//     Term 19 (AT2200-0500)/CC Outputs/Current setpoint value Ch.8 <-> Data Pointer/CurrentSetpointValues[7]
//     Term 19 (AT2200-0500)/CC Outputs/Current setpoint value Ch.9 <-> Data Pointer/CurrentSetpointValues[8]
//     Term 19 (AT2200-0500)/LFB Inputs/BinaryData <-> Data Pointer/HallSensorValues
//   Device 20 <-> TcCOM Objects/XTS ProcessingUnit 1/Part 1/Module 16
//     Term 20 (AT2200-0500)/CC Inputs/Current actual value Ch.1 <-> Data Pointer/CurrentActualValues[0]
//     Term 20 (AT2200-0500)/CC Inputs/Current actual value Ch.10 <-> Data Pointer/CurrentActualValues[9]
//     Term 20 (AT2200-0500)/CC Inputs/Current actual value Ch.11 <-> Data Pointer/CurrentActualValues[10]
//     Term 20 (AT2200-0500)/CC Inputs/Current actual value Ch.12 <-> Data Pointer/CurrentActualValues[11]
//     Term 20 (AT2200-0500)/CC Inputs/Current actual value Ch.13 <-> Data Pointer/CurrentActualValues[12]
//     Term 20 (AT2200-0500)/CC Inputs/Current actual value Ch.14 <-> Data Pointer/CurrentActualValues[13]
//     Term 20 (AT2200-0500)/CC Inputs/Current actual value Ch.15 <-> Data Pointer/CurrentActualValues[14]
//     Term 20 (AT2200-0500)/CC Inputs/Current actual value Ch.16 <-> Data Pointer/CurrentActualValues[15]
//     Term 20 (AT2200-0500)/CC Inputs/Current actual value Ch.17 <-> Data Pointer/CurrentActualValues[16]
//     Term 20 (AT2200-0500)/CC Inputs/Current actual value Ch.18 <-> Data Pointer/CurrentActualValues[17]
//     Term 20 (AT2200-0500)/CC Inputs/Current actual value Ch.19 <-> Data Pointer/CurrentActualValues[18]
//     Term 20 (AT2200-0500)/CC Inputs/Current actual value Ch.2 <-> Data Pointer/CurrentActualValues[1]
//     Term 20 (AT2200-0500)/CC Inputs/Current actual value Ch.20 <-> Data Pointer/CurrentActualValues[19]
//     Term 20 (AT2200-0500)/CC Inputs/Current actual value Ch.21 <-> Data Pointer/CurrentActualValues[20]
//     Term 20 (AT2200-0500)/CC Inputs/Current actual value Ch.22 <-> Data Pointer/CurrentActualValues[21]
//     Term 20 (AT2200-0500)/CC Inputs/Current actual value Ch.23 <-> Data Pointer/CurrentActualValues[22]
//     Term 20 (AT2200-0500)/CC Inputs/Current actual value Ch.24 <-> Data Pointer/CurrentActualValues[23]
//     Term 20 (AT2200-0500)/CC Inputs/Current actual value Ch.25 <-> Data Pointer/CurrentActualValues[24]
//     Term 20 (AT2200-0500)/CC Inputs/Current actual value Ch.26 <-> Data Pointer/CurrentActualValues[25]
//     Term 20 (AT2200-0500)/CC Inputs/Current actual value Ch.27 <-> Data Pointer/CurrentActualValues[26]
//     Term 20 (AT2200-0500)/CC Inputs/Current actual value Ch.28 <-> Data Pointer/CurrentActualValues[27]
//     Term 20 (AT2200-0500)/CC Inputs/Current actual value Ch.29 <-> Data Pointer/CurrentActualValues[28]
//     Term 20 (AT2200-0500)/CC Inputs/Current actual value Ch.3 <-> Data Pointer/CurrentActualValues[2]
//     Term 20 (AT2200-0500)/CC Inputs/Current actual value Ch.30 <-> Data Pointer/CurrentActualValues[29]
//     Term 20 (AT2200-0500)/CC Inputs/Current actual value Ch.4 <-> Data Pointer/CurrentActualValues[3]
//     Term 20 (AT2200-0500)/CC Inputs/Current actual value Ch.5 <-> Data Pointer/CurrentActualValues[4]
//     Term 20 (AT2200-0500)/CC Inputs/Current actual value Ch.6 <-> Data Pointer/CurrentActualValues[5]
//     Term 20 (AT2200-0500)/CC Inputs/Current actual value Ch.7 <-> Data Pointer/CurrentActualValues[6]
//     Term 20 (AT2200-0500)/CC Inputs/Current actual value Ch.8 <-> Data Pointer/CurrentActualValues[7]
//     Term 20 (AT2200-0500)/CC Inputs/Current actual value Ch.9 <-> Data Pointer/CurrentActualValues[8]
//     Term 20 (AT2200-0500)/CC Inputs/Status <-> Data Pointer/Status
//     Term 20 (AT2200-0500)/CC Outputs/Control <-> Data Pointer/Control
//     Term 20 (AT2200-0500)/CC Outputs/Current setpoint value Ch.1 <-> Data Pointer/CurrentSetpointValues[0]
//     Term 20 (AT2200-0500)/CC Outputs/Current setpoint value Ch.10 <-> Data Pointer/CurrentSetpointValues[9]
//     Term 20 (AT2200-0500)/CC Outputs/Current setpoint value Ch.11 <-> Data Pointer/CurrentSetpointValues[10]
//     Term 20 (AT2200-0500)/CC Outputs/Current setpoint value Ch.12 <-> Data Pointer/CurrentSetpointValues[11]
//     Term 20 (AT2200-0500)/CC Outputs/Current setpoint value Ch.13 <-> Data Pointer/CurrentSetpointValues[12]
//     Term 20 (AT2200-0500)/CC Outputs/Current setpoint value Ch.14 <-> Data Pointer/CurrentSetpointValues[13]
//     Term 20 (AT2200-0500)/CC Outputs/Current setpoint value Ch.15 <-> Data Pointer/CurrentSetpointValues[14]
//     Term 20 (AT2200-0500)/CC Outputs/Current setpoint value Ch.16 <-> Data Pointer/CurrentSetpointValues[15]
//     Term 20 (AT2200-0500)/CC Outputs/Current setpoint value Ch.17 <-> Data Pointer/CurrentSetpointValues[16]
//     Term 20 (AT2200-0500)/CC Outputs/Current setpoint value Ch.18 <-> Data Pointer/CurrentSetpointValues[17]
//     Term 20 (AT2200-0500)/CC Outputs/Current setpoint value Ch.19 <-> Data Pointer/CurrentSetpointValues[18]
//     Term 20 (AT2200-0500)/CC Outputs/Current setpoint value Ch.2 <-> Data Pointer/CurrentSetpointValues[1]
//     Term 20 (AT2200-0500)/CC Outputs/Current setpoint value Ch.20 <-> Data Pointer/CurrentSetpointValues[19]
//     Term 20 (AT2200-0500)/CC Outputs/Current setpoint value Ch.21 <-> Data Pointer/CurrentSetpointValues[20]
//     Term 20 (AT2200-0500)/CC Outputs/Current setpoint value Ch.22 <-> Data Pointer/CurrentSetpointValues[21]
//     Term 20 (AT2200-0500)/CC Outputs/Current setpoint value Ch.23 <-> Data Pointer/CurrentSetpointValues[22]
//     Term 20 (AT2200-0500)/CC Outputs/Current setpoint value Ch.24 <-> Data Pointer/CurrentSetpointValues[23]
//     Term 20 (AT2200-0500)/CC Outputs/Current setpoint value Ch.25 <-> Data Pointer/CurrentSetpointValues[24]
//     Term 20 (AT2200-0500)/CC Outputs/Current setpoint value Ch.26 <-> Data Pointer/CurrentSetpointValues[25]
//     Term 20 (AT2200-0500)/CC Outputs/Current setpoint value Ch.27 <-> Data Pointer/CurrentSetpointValues[26]
//     Term 20 (AT2200-0500)/CC Outputs/Current setpoint value Ch.28 <-> Data Pointer/CurrentSetpointValues[27]
//     Term 20 (AT2200-0500)/CC Outputs/Current setpoint value Ch.29 <-> Data Pointer/CurrentSetpointValues[28]
//     Term 20 (AT2200-0500)/CC Outputs/Current setpoint value Ch.3 <-> Data Pointer/CurrentSetpointValues[2]
//     Term 20 (AT2200-0500)/CC Outputs/Current setpoint value Ch.30 <-> Data Pointer/CurrentSetpointValues[29]
//     Term 20 (AT2200-0500)/CC Outputs/Current setpoint value Ch.4 <-> Data Pointer/CurrentSetpointValues[3]
//     Term 20 (AT2200-0500)/CC Outputs/Current setpoint value Ch.5 <-> Data Pointer/CurrentSetpointValues[4]
//     Term 20 (AT2200-0500)/CC Outputs/Current setpoint value Ch.6 <-> Data Pointer/CurrentSetpointValues[5]
//     Term 20 (AT2200-0500)/CC Outputs/Current setpoint value Ch.7 <-> Data Pointer/CurrentSetpointValues[6]
//     Term 20 (AT2200-0500)/CC Outputs/Current setpoint value Ch.8 <-> Data Pointer/CurrentSetpointValues[7]
//     Term 20 (AT2200-0500)/CC Outputs/Current setpoint value Ch.9 <-> Data Pointer/CurrentSetpointValues[8]
//     Term 20 (AT2200-0500)/LFB Inputs/BinaryData <-> Data Pointer/HallSensorValues
//   Device 21 <-> TcCOM Objects/XTS ProcessingUnit 1/Part 1/Module 17
//     Term 21 (AT2202-0500)/CC Inputs/Current actual value Ch.1 <-> Data Pointer/CurrentActualValues[0]
//     Term 21 (AT2202-0500)/CC Inputs/Current actual value Ch.10 <-> Data Pointer/CurrentActualValues[9]
//     Term 21 (AT2202-0500)/CC Inputs/Current actual value Ch.11 <-> Data Pointer/CurrentActualValues[10]
//     Term 21 (AT2202-0500)/CC Inputs/Current actual value Ch.12 <-> Data Pointer/CurrentActualValues[11]
//     Term 21 (AT2202-0500)/CC Inputs/Current actual value Ch.13 <-> Data Pointer/CurrentActualValues[12]
//     Term 21 (AT2202-0500)/CC Inputs/Current actual value Ch.14 <-> Data Pointer/CurrentActualValues[13]
//     Term 21 (AT2202-0500)/CC Inputs/Current actual value Ch.15 <-> Data Pointer/CurrentActualValues[14]
//     Term 21 (AT2202-0500)/CC Inputs/Current actual value Ch.16 <-> Data Pointer/CurrentActualValues[15]
//     Term 21 (AT2202-0500)/CC Inputs/Current actual value Ch.17 <-> Data Pointer/CurrentActualValues[16]
//     Term 21 (AT2202-0500)/CC Inputs/Current actual value Ch.18 <-> Data Pointer/CurrentActualValues[17]
//     Term 21 (AT2202-0500)/CC Inputs/Current actual value Ch.19 <-> Data Pointer/CurrentActualValues[18]
//     Term 21 (AT2202-0500)/CC Inputs/Current actual value Ch.2 <-> Data Pointer/CurrentActualValues[1]
//     Term 21 (AT2202-0500)/CC Inputs/Current actual value Ch.20 <-> Data Pointer/CurrentActualValues[19]
//     Term 21 (AT2202-0500)/CC Inputs/Current actual value Ch.21 <-> Data Pointer/CurrentActualValues[20]
//     Term 21 (AT2202-0500)/CC Inputs/Current actual value Ch.22 <-> Data Pointer/CurrentActualValues[21]
//     Term 21 (AT2202-0500)/CC Inputs/Current actual value Ch.23 <-> Data Pointer/CurrentActualValues[22]
//     Term 21 (AT2202-0500)/CC Inputs/Current actual value Ch.24 <-> Data Pointer/CurrentActualValues[23]
//     Term 21 (AT2202-0500)/CC Inputs/Current actual value Ch.25 <-> Data Pointer/CurrentActualValues[24]
//     Term 21 (AT2202-0500)/CC Inputs/Current actual value Ch.26 <-> Data Pointer/CurrentActualValues[25]
//     Term 21 (AT2202-0500)/CC Inputs/Current actual value Ch.27 <-> Data Pointer/CurrentActualValues[26]
//     Term 21 (AT2202-0500)/CC Inputs/Current actual value Ch.28 <-> Data Pointer/CurrentActualValues[27]
//     Term 21 (AT2202-0500)/CC Inputs/Current actual value Ch.29 <-> Data Pointer/CurrentActualValues[28]
//     Term 21 (AT2202-0500)/CC Inputs/Current actual value Ch.3 <-> Data Pointer/CurrentActualValues[2]
//     Term 21 (AT2202-0500)/CC Inputs/Current actual value Ch.30 <-> Data Pointer/CurrentActualValues[29]
//     Term 21 (AT2202-0500)/CC Inputs/Current actual value Ch.4 <-> Data Pointer/CurrentActualValues[3]
//     Term 21 (AT2202-0500)/CC Inputs/Current actual value Ch.5 <-> Data Pointer/CurrentActualValues[4]
//     Term 21 (AT2202-0500)/CC Inputs/Current actual value Ch.6 <-> Data Pointer/CurrentActualValues[5]
//     Term 21 (AT2202-0500)/CC Inputs/Current actual value Ch.7 <-> Data Pointer/CurrentActualValues[6]
//     Term 21 (AT2202-0500)/CC Inputs/Current actual value Ch.8 <-> Data Pointer/CurrentActualValues[7]
//     Term 21 (AT2202-0500)/CC Inputs/Current actual value Ch.9 <-> Data Pointer/CurrentActualValues[8]
//     Term 21 (AT2202-0500)/CC Inputs/Status <-> Data Pointer/Status
//     Term 21 (AT2202-0500)/CC Outputs/Control <-> Data Pointer/Control
//     Term 21 (AT2202-0500)/CC Outputs/Current setpoint value Ch.1 <-> Data Pointer/CurrentSetpointValues[0]
//     Term 21 (AT2202-0500)/CC Outputs/Current setpoint value Ch.10 <-> Data Pointer/CurrentSetpointValues[9]
//     Term 21 (AT2202-0500)/CC Outputs/Current setpoint value Ch.11 <-> Data Pointer/CurrentSetpointValues[10]
//     Term 21 (AT2202-0500)/CC Outputs/Current setpoint value Ch.12 <-> Data Pointer/CurrentSetpointValues[11]
//     Term 21 (AT2202-0500)/CC Outputs/Current setpoint value Ch.13 <-> Data Pointer/CurrentSetpointValues[12]
//     Term 21 (AT2202-0500)/CC Outputs/Current setpoint value Ch.14 <-> Data Pointer/CurrentSetpointValues[13]
//     Term 21 (AT2202-0500)/CC Outputs/Current setpoint value Ch.15 <-> Data Pointer/CurrentSetpointValues[14]
//     Term 21 (AT2202-0500)/CC Outputs/Current setpoint value Ch.16 <-> Data Pointer/CurrentSetpointValues[15]
//     Term 21 (AT2202-0500)/CC Outputs/Current setpoint value Ch.17 <-> Data Pointer/CurrentSetpointValues[16]
//     Term 21 (AT2202-0500)/CC Outputs/Current setpoint value Ch.18 <-> Data Pointer/CurrentSetpointValues[17]
//     Term 21 (AT2202-0500)/CC Outputs/Current setpoint value Ch.19 <-> Data Pointer/CurrentSetpointValues[18]
//     Term 21 (AT2202-0500)/CC Outputs/Current setpoint value Ch.2 <-> Data Pointer/CurrentSetpointValues[1]
//     Term 21 (AT2202-0500)/CC Outputs/Current setpoint value Ch.20 <-> Data Pointer/CurrentSetpointValues[19]
//     Term 21 (AT2202-0500)/CC Outputs/Current setpoint value Ch.21 <-> Data Pointer/CurrentSetpointValues[20]
//     Term 21 (AT2202-0500)/CC Outputs/Current setpoint value Ch.22 <-> Data Pointer/CurrentSetpointValues[21]
//     Term 21 (AT2202-0500)/CC Outputs/Current setpoint value Ch.23 <-> Data Pointer/CurrentSetpointValues[22]
//     Term 21 (AT2202-0500)/CC Outputs/Current setpoint value Ch.24 <-> Data Pointer/CurrentSetpointValues[23]
//     Term 21 (AT2202-0500)/CC Outputs/Current setpoint value Ch.25 <-> Data Pointer/CurrentSetpointValues[24]
//     Term 21 (AT2202-0500)/CC Outputs/Current setpoint value Ch.26 <-> Data Pointer/CurrentSetpointValues[25]
//     Term 21 (AT2202-0500)/CC Outputs/Current setpoint value Ch.27 <-> Data Pointer/CurrentSetpointValues[26]
//     Term 21 (AT2202-0500)/CC Outputs/Current setpoint value Ch.28 <-> Data Pointer/CurrentSetpointValues[27]
//     Term 21 (AT2202-0500)/CC Outputs/Current setpoint value Ch.29 <-> Data Pointer/CurrentSetpointValues[28]
//     Term 21 (AT2202-0500)/CC Outputs/Current setpoint value Ch.3 <-> Data Pointer/CurrentSetpointValues[2]
//     Term 21 (AT2202-0500)/CC Outputs/Current setpoint value Ch.30 <-> Data Pointer/CurrentSetpointValues[29]
//     Term 21 (AT2202-0500)/CC Outputs/Current setpoint value Ch.4 <-> Data Pointer/CurrentSetpointValues[3]
//     Term 21 (AT2202-0500)/CC Outputs/Current setpoint value Ch.5 <-> Data Pointer/CurrentSetpointValues[4]
//     Term 21 (AT2202-0500)/CC Outputs/Current setpoint value Ch.6 <-> Data Pointer/CurrentSetpointValues[5]
//     Term 21 (AT2202-0500)/CC Outputs/Current setpoint value Ch.7 <-> Data Pointer/CurrentSetpointValues[6]
//     Term 21 (AT2202-0500)/CC Outputs/Current setpoint value Ch.8 <-> Data Pointer/CurrentSetpointValues[7]
//     Term 21 (AT2202-0500)/CC Outputs/Current setpoint value Ch.9 <-> Data Pointer/CurrentSetpointValues[8]
//     Term 21 (AT2202-0500)/LFB Inputs/BinaryData <-> Data Pointer/HallSensorValues
//   Device 21 <-> TcCOM Objects/XTS ProcessingUnit 1/Part 1/Module 18
//     Term 22 (AT2200-0500)/CC Inputs/Current actual value Ch.1 <-> Data Pointer/CurrentActualValues[0]
//     Term 22 (AT2200-0500)/CC Inputs/Current actual value Ch.10 <-> Data Pointer/CurrentActualValues[9]
//     Term 22 (AT2200-0500)/CC Inputs/Current actual value Ch.11 <-> Data Pointer/CurrentActualValues[10]
//     Term 22 (AT2200-0500)/CC Inputs/Current actual value Ch.12 <-> Data Pointer/CurrentActualValues[11]
//     Term 22 (AT2200-0500)/CC Inputs/Current actual value Ch.13 <-> Data Pointer/CurrentActualValues[12]
//     Term 22 (AT2200-0500)/CC Inputs/Current actual value Ch.14 <-> Data Pointer/CurrentActualValues[13]
//     Term 22 (AT2200-0500)/CC Inputs/Current actual value Ch.15 <-> Data Pointer/CurrentActualValues[14]
//     Term 22 (AT2200-0500)/CC Inputs/Current actual value Ch.16 <-> Data Pointer/CurrentActualValues[15]
//     Term 22 (AT2200-0500)/CC Inputs/Current actual value Ch.17 <-> Data Pointer/CurrentActualValues[16]
//     Term 22 (AT2200-0500)/CC Inputs/Current actual value Ch.18 <-> Data Pointer/CurrentActualValues[17]
//     Term 22 (AT2200-0500)/CC Inputs/Current actual value Ch.19 <-> Data Pointer/CurrentActualValues[18]
//     Term 22 (AT2200-0500)/CC Inputs/Current actual value Ch.2 <-> Data Pointer/CurrentActualValues[1]
//     Term 22 (AT2200-0500)/CC Inputs/Current actual value Ch.20 <-> Data Pointer/CurrentActualValues[19]
//     Term 22 (AT2200-0500)/CC Inputs/Current actual value Ch.21 <-> Data Pointer/CurrentActualValues[20]
//     Term 22 (AT2200-0500)/CC Inputs/Current actual value Ch.22 <-> Data Pointer/CurrentActualValues[21]
//     Term 22 (AT2200-0500)/CC Inputs/Current actual value Ch.23 <-> Data Pointer/CurrentActualValues[22]
//     Term 22 (AT2200-0500)/CC Inputs/Current actual value Ch.24 <-> Data Pointer/CurrentActualValues[23]
//     Term 22 (AT2200-0500)/CC Inputs/Current actual value Ch.25 <-> Data Pointer/CurrentActualValues[24]
//     Term 22 (AT2200-0500)/CC Inputs/Current actual value Ch.26 <-> Data Pointer/CurrentActualValues[25]
//     Term 22 (AT2200-0500)/CC Inputs/Current actual value Ch.27 <-> Data Pointer/CurrentActualValues[26]
//     Term 22 (AT2200-0500)/CC Inputs/Current actual value Ch.28 <-> Data Pointer/CurrentActualValues[27]
//     Term 22 (AT2200-0500)/CC Inputs/Current actual value Ch.29 <-> Data Pointer/CurrentActualValues[28]
//     Term 22 (AT2200-0500)/CC Inputs/Current actual value Ch.3 <-> Data Pointer/CurrentActualValues[2]
//     Term 22 (AT2200-0500)/CC Inputs/Current actual value Ch.30 <-> Data Pointer/CurrentActualValues[29]
//     Term 22 (AT2200-0500)/CC Inputs/Current actual value Ch.4 <-> Data Pointer/CurrentActualValues[3]
//     Term 22 (AT2200-0500)/CC Inputs/Current actual value Ch.5 <-> Data Pointer/CurrentActualValues[4]
//     Term 22 (AT2200-0500)/CC Inputs/Current actual value Ch.6 <-> Data Pointer/CurrentActualValues[5]
//     Term 22 (AT2200-0500)/CC Inputs/Current actual value Ch.7 <-> Data Pointer/CurrentActualValues[6]
//     Term 22 (AT2200-0500)/CC Inputs/Current actual value Ch.8 <-> Data Pointer/CurrentActualValues[7]
//     Term 22 (AT2200-0500)/CC Inputs/Current actual value Ch.9 <-> Data Pointer/CurrentActualValues[8]
//     Term 22 (AT2200-0500)/CC Inputs/Status <-> Data Pointer/Status
//     Term 22 (AT2200-0500)/CC Outputs/Control <-> Data Pointer/Control
//     Term 22 (AT2200-0500)/CC Outputs/Current setpoint value Ch.1 <-> Data Pointer/CurrentSetpointValues[0]
//     Term 22 (AT2200-0500)/CC Outputs/Current setpoint value Ch.10 <-> Data Pointer/CurrentSetpointValues[9]
//     Term 22 (AT2200-0500)/CC Outputs/Current setpoint value Ch.11 <-> Data Pointer/CurrentSetpointValues[10]
//     Term 22 (AT2200-0500)/CC Outputs/Current setpoint value Ch.12 <-> Data Pointer/CurrentSetpointValues[11]
//     Term 22 (AT2200-0500)/CC Outputs/Current setpoint value Ch.13 <-> Data Pointer/CurrentSetpointValues[12]
//     Term 22 (AT2200-0500)/CC Outputs/Current setpoint value Ch.14 <-> Data Pointer/CurrentSetpointValues[13]
//     Term 22 (AT2200-0500)/CC Outputs/Current setpoint value Ch.15 <-> Data Pointer/CurrentSetpointValues[14]
//     Term 22 (AT2200-0500)/CC Outputs/Current setpoint value Ch.16 <-> Data Pointer/CurrentSetpointValues[15]
//     Term 22 (AT2200-0500)/CC Outputs/Current setpoint value Ch.17 <-> Data Pointer/CurrentSetpointValues[16]
//     Term 22 (AT2200-0500)/CC Outputs/Current setpoint value Ch.18 <-> Data Pointer/CurrentSetpointValues[17]
//     Term 22 (AT2200-0500)/CC Outputs/Current setpoint value Ch.19 <-> Data Pointer/CurrentSetpointValues[18]
//     Term 22 (AT2200-0500)/CC Outputs/Current setpoint value Ch.2 <-> Data Pointer/CurrentSetpointValues[1]
//     Term 22 (AT2200-0500)/CC Outputs/Current setpoint value Ch.20 <-> Data Pointer/CurrentSetpointValues[19]
//     Term 22 (AT2200-0500)/CC Outputs/Current setpoint value Ch.21 <-> Data Pointer/CurrentSetpointValues[20]
//     Term 22 (AT2200-0500)/CC Outputs/Current setpoint value Ch.22 <-> Data Pointer/CurrentSetpointValues[21]
//     Term 22 (AT2200-0500)/CC Outputs/Current setpoint value Ch.23 <-> Data Pointer/CurrentSetpointValues[22]
//     Term 22 (AT2200-0500)/CC Outputs/Current setpoint value Ch.24 <-> Data Pointer/CurrentSetpointValues[23]
//     Term 22 (AT2200-0500)/CC Outputs/Current setpoint value Ch.25 <-> Data Pointer/CurrentSetpointValues[24]
//     Term 22 (AT2200-0500)/CC Outputs/Current setpoint value Ch.26 <-> Data Pointer/CurrentSetpointValues[25]
//     Term 22 (AT2200-0500)/CC Outputs/Current setpoint value Ch.27 <-> Data Pointer/CurrentSetpointValues[26]
//     Term 22 (AT2200-0500)/CC Outputs/Current setpoint value Ch.28 <-> Data Pointer/CurrentSetpointValues[27]
//     Term 22 (AT2200-0500)/CC Outputs/Current setpoint value Ch.29 <-> Data Pointer/CurrentSetpointValues[28]
//     Term 22 (AT2200-0500)/CC Outputs/Current setpoint value Ch.3 <-> Data Pointer/CurrentSetpointValues[2]
//     Term 22 (AT2200-0500)/CC Outputs/Current setpoint value Ch.30 <-> Data Pointer/CurrentSetpointValues[29]
//     Term 22 (AT2200-0500)/CC Outputs/Current setpoint value Ch.4 <-> Data Pointer/CurrentSetpointValues[3]
//     Term 22 (AT2200-0500)/CC Outputs/Current setpoint value Ch.5 <-> Data Pointer/CurrentSetpointValues[4]
//     Term 22 (AT2200-0500)/CC Outputs/Current setpoint value Ch.6 <-> Data Pointer/CurrentSetpointValues[5]
//     Term 22 (AT2200-0500)/CC Outputs/Current setpoint value Ch.7 <-> Data Pointer/CurrentSetpointValues[6]
//     Term 22 (AT2200-0500)/CC Outputs/Current setpoint value Ch.8 <-> Data Pointer/CurrentSetpointValues[7]
//     Term 22 (AT2200-0500)/CC Outputs/Current setpoint value Ch.9 <-> Data Pointer/CurrentSetpointValues[8]
//     Term 22 (AT2200-0500)/LFB Inputs/BinaryData <-> Data Pointer/HallSensorValues
//   Device 21 <-> TcCOM Objects/XTS ProcessingUnit 1/Part 1/Module 19
//     Term 23 (AT2000-0250)/CC Inputs/Current actual value Ch.1 <-> Data Pointer/CurrentActualValues[0]
//     Term 23 (AT2000-0250)/CC Inputs/Current actual value Ch.10 <-> Data Pointer/CurrentActualValues[9]
//     Term 23 (AT2000-0250)/CC Inputs/Current actual value Ch.11 <-> Data Pointer/CurrentActualValues[10]
//     Term 23 (AT2000-0250)/CC Inputs/Current actual value Ch.12 <-> Data Pointer/CurrentActualValues[11]
//     Term 23 (AT2000-0250)/CC Inputs/Current actual value Ch.13 <-> Data Pointer/CurrentActualValues[12]
//     Term 23 (AT2000-0250)/CC Inputs/Current actual value Ch.14 <-> Data Pointer/CurrentActualValues[13]
//     Term 23 (AT2000-0250)/CC Inputs/Current actual value Ch.15 <-> Data Pointer/CurrentActualValues[14]
//     Term 23 (AT2000-0250)/CC Inputs/Current actual value Ch.2 <-> Data Pointer/CurrentActualValues[1]
//     Term 23 (AT2000-0250)/CC Inputs/Current actual value Ch.3 <-> Data Pointer/CurrentActualValues[2]
//     Term 23 (AT2000-0250)/CC Inputs/Current actual value Ch.4 <-> Data Pointer/CurrentActualValues[3]
//     Term 23 (AT2000-0250)/CC Inputs/Current actual value Ch.5 <-> Data Pointer/CurrentActualValues[4]
//     Term 23 (AT2000-0250)/CC Inputs/Current actual value Ch.6 <-> Data Pointer/CurrentActualValues[5]
//     Term 23 (AT2000-0250)/CC Inputs/Current actual value Ch.7 <-> Data Pointer/CurrentActualValues[6]
//     Term 23 (AT2000-0250)/CC Inputs/Current actual value Ch.8 <-> Data Pointer/CurrentActualValues[7]
//     Term 23 (AT2000-0250)/CC Inputs/Current actual value Ch.9 <-> Data Pointer/CurrentActualValues[8]
//     Term 23 (AT2000-0250)/CC Inputs/Status <-> Data Pointer/Status
//     Term 23 (AT2000-0250)/CC Outputs/Control <-> Data Pointer/Control
//     Term 23 (AT2000-0250)/CC Outputs/Current setpoint value Ch.1 <-> Data Pointer/CurrentSetpointValues[0]
//     Term 23 (AT2000-0250)/CC Outputs/Current setpoint value Ch.10 <-> Data Pointer/CurrentSetpointValues[9]
//     Term 23 (AT2000-0250)/CC Outputs/Current setpoint value Ch.11 <-> Data Pointer/CurrentSetpointValues[10]
//     Term 23 (AT2000-0250)/CC Outputs/Current setpoint value Ch.12 <-> Data Pointer/CurrentSetpointValues[11]
//     Term 23 (AT2000-0250)/CC Outputs/Current setpoint value Ch.13 <-> Data Pointer/CurrentSetpointValues[12]
//     Term 23 (AT2000-0250)/CC Outputs/Current setpoint value Ch.14 <-> Data Pointer/CurrentSetpointValues[13]
//     Term 23 (AT2000-0250)/CC Outputs/Current setpoint value Ch.15 <-> Data Pointer/CurrentSetpointValues[14]
//     Term 23 (AT2000-0250)/CC Outputs/Current setpoint value Ch.2 <-> Data Pointer/CurrentSetpointValues[1]
//     Term 23 (AT2000-0250)/CC Outputs/Current setpoint value Ch.3 <-> Data Pointer/CurrentSetpointValues[2]
//     Term 23 (AT2000-0250)/CC Outputs/Current setpoint value Ch.4 <-> Data Pointer/CurrentSetpointValues[3]
//     Term 23 (AT2000-0250)/CC Outputs/Current setpoint value Ch.5 <-> Data Pointer/CurrentSetpointValues[4]
//     Term 23 (AT2000-0250)/CC Outputs/Current setpoint value Ch.6 <-> Data Pointer/CurrentSetpointValues[5]
//     Term 23 (AT2000-0250)/CC Outputs/Current setpoint value Ch.7 <-> Data Pointer/CurrentSetpointValues[6]
//     Term 23 (AT2000-0250)/CC Outputs/Current setpoint value Ch.8 <-> Data Pointer/CurrentSetpointValues[7]
//     Term 23 (AT2000-0250)/CC Outputs/Current setpoint value Ch.9 <-> Data Pointer/CurrentSetpointValues[8]
//     Term 23 (AT2000-0250)/Term 24 (AT2000-5250)/FB Inputs/Value Channel 01 <-> Data Pointer/RawPositionValues[0]
//     Term 23 (AT2000-0250)/Term 24 (AT2000-5250)/FB Inputs/Value Channel 02 <-> Data Pointer/RawPositionValues[1]
//     Term 23 (AT2000-0250)/Term 24 (AT2000-5250)/FB Inputs/Value Channel 03 <-> Data Pointer/RawPositionValues[2]
//     Term 23 (AT2000-0250)/Term 24 (AT2000-5250)/FB Inputs/Value Channel 04 <-> Data Pointer/RawPositionValues[3]
//     Term 23 (AT2000-0250)/Term 24 (AT2000-5250)/FB Inputs/Value Channel 05 <-> Data Pointer/RawPositionValues[4]
//     Term 23 (AT2000-0250)/Term 24 (AT2000-5250)/FB Inputs/Value Channel 06 <-> Data Pointer/RawPositionValues[5]
//     Term 23 (AT2000-0250)/Term 24 (AT2000-5250)/FB Inputs/Value Channel 07 <-> Data Pointer/RawPositionValues[6]
//     Term 23 (AT2000-0250)/Term 24 (AT2000-5250)/FB Inputs/Value Channel 08 <-> Data Pointer/RawPositionValues[7]
//     Term 23 (AT2000-0250)/Term 24 (AT2000-5250)/FB Inputs/Value Channel 09 <-> Data Pointer/RawPositionValues[8]
//     Term 23 (AT2000-0250)/Term 24 (AT2000-5250)/FB Inputs/Value Channel 10 <-> Data Pointer/RawPositionValues[9]
//     Term 23 (AT2000-0250)/Term 24 (AT2000-5250)/FB Inputs/Value Channel 11 <-> Data Pointer/RawPositionValues[10]
//     Term 23 (AT2000-0250)/Term 24 (AT2000-5250)/FB Inputs/Value Channel 12 <-> Data Pointer/RawPositionValues[11]
//     Term 23 (AT2000-0250)/Term 24 (AT2000-5250)/FB Inputs/Value Channel 13 <-> Data Pointer/RawPositionValues[12]
//     Term 23 (AT2000-0250)/Term 24 (AT2000-5250)/FB Inputs/Value Channel 14 <-> Data Pointer/RawPositionValues[13]
//     Term 23 (AT2000-0250)/Term 24 (AT2000-5250)/FB Inputs/Value Channel 15 <-> Data Pointer/RawPositionValues[14]
//     Term 23 (AT2000-0250)/Term 24 (AT2000-5250)/FB Inputs/Value Channel 16 <-> Data Pointer/RawPositionValues[15]
//     Term 23 (AT2000-0250)/Term 24 (AT2000-5250)/FB Inputs/Value Channel 17 <-> Data Pointer/RawPositionValues[16]
//     Term 23 (AT2000-0250)/Term 24 (AT2000-5250)/FB Inputs/Value Channel 18 <-> Data Pointer/RawPositionValues[17]
//     Term 23 (AT2000-0250)/Term 24 (AT2000-5250)/FB Inputs/Value Channel 19 <-> Data Pointer/RawPositionValues[18]
//     Term 23 (AT2000-0250)/Term 24 (AT2000-5250)/FB Inputs/Value Channel 20 <-> Data Pointer/RawPositionValues[19]
//     Term 23 (AT2000-0250)/Term 24 (AT2000-5250)/FB Inputs/Value Channel 21 <-> Data Pointer/RawPositionValues[20]
//     Term 23 (AT2000-0250)/Term 24 (AT2000-5250)/FB Inputs/Value Channel 22 <-> Data Pointer/RawPositionValues[21]
//     Term 23 (AT2000-0250)/Term 24 (AT2000-5250)/FB Inputs/Value Channel 23 <-> Data Pointer/RawPositionValues[22]
//     Term 23 (AT2000-0250)/Term 24 (AT2000-5250)/FB Inputs/Value Channel 24 <-> Data Pointer/RawPositionValues[23]
//     Term 23 (AT2000-0250)/Term 24 (AT2000-5250)/FB Inputs/Value Channel 25 <-> Data Pointer/RawPositionValues[24]
//     Term 23 (AT2000-0250)/Term 24 (AT2000-5250)/FB Inputs/Value Channel 26 <-> Data Pointer/RawPositionValues[25]
//     Term 23 (AT2000-0250)/Term 24 (AT2000-5250)/FB Inputs/Value Channel 27 <-> Data Pointer/RawPositionValues[26]
//     Term 23 (AT2000-0250)/Term 24 (AT2000-5250)/FB Inputs/Value Channel 28 <-> Data Pointer/RawPositionValues[27]
//     Term 23 (AT2000-0250)/Term 24 (AT2000-5250)/FB Inputs/Value Channel 29 <-> Data Pointer/RawPositionValues[28]
//     Term 23 (AT2000-0250)/Term 24 (AT2000-5250)/FB Inputs/Value Channel 30 <-> Data Pointer/RawPositionValues[29]
//     Term 23 (AT2000-0250)/Term 24 (AT2000-5250)/FB Inputs/Value Channel 31 <-> Data Pointer/RawPositionValues[30]
//     Term 23 (AT2000-0250)/Term 24 (AT2000-5250)/FB Inputs/Value Channel 32 <-> Data Pointer/RawPositionValues[31]
//   Device 22 <-> TcCOM Objects/XTS ProcessingUnit 1/Part 1/Module 20
//     Term 25 (AT2002-0250)/CC Inputs/Current actual value Ch.1 <-> Data Pointer/CurrentActualValues[0]
//     Term 25 (AT2002-0250)/CC Inputs/Current actual value Ch.10 <-> Data Pointer/CurrentActualValues[9]
//     Term 25 (AT2002-0250)/CC Inputs/Current actual value Ch.11 <-> Data Pointer/CurrentActualValues[10]
//     Term 25 (AT2002-0250)/CC Inputs/Current actual value Ch.12 <-> Data Pointer/CurrentActualValues[11]
//     Term 25 (AT2002-0250)/CC Inputs/Current actual value Ch.13 <-> Data Pointer/CurrentActualValues[12]
//     Term 25 (AT2002-0250)/CC Inputs/Current actual value Ch.14 <-> Data Pointer/CurrentActualValues[13]
//     Term 25 (AT2002-0250)/CC Inputs/Current actual value Ch.15 <-> Data Pointer/CurrentActualValues[14]
//     Term 25 (AT2002-0250)/CC Inputs/Current actual value Ch.2 <-> Data Pointer/CurrentActualValues[1]
//     Term 25 (AT2002-0250)/CC Inputs/Current actual value Ch.3 <-> Data Pointer/CurrentActualValues[2]
//     Term 25 (AT2002-0250)/CC Inputs/Current actual value Ch.4 <-> Data Pointer/CurrentActualValues[3]
//     Term 25 (AT2002-0250)/CC Inputs/Current actual value Ch.5 <-> Data Pointer/CurrentActualValues[4]
//     Term 25 (AT2002-0250)/CC Inputs/Current actual value Ch.6 <-> Data Pointer/CurrentActualValues[5]
//     Term 25 (AT2002-0250)/CC Inputs/Current actual value Ch.7 <-> Data Pointer/CurrentActualValues[6]
//     Term 25 (AT2002-0250)/CC Inputs/Current actual value Ch.8 <-> Data Pointer/CurrentActualValues[7]
//     Term 25 (AT2002-0250)/CC Inputs/Current actual value Ch.9 <-> Data Pointer/CurrentActualValues[8]
//     Term 25 (AT2002-0250)/CC Inputs/Status <-> Data Pointer/Status
//     Term 25 (AT2002-0250)/CC Outputs/Control <-> Data Pointer/Control
//     Term 25 (AT2002-0250)/CC Outputs/Current setpoint value Ch.1 <-> Data Pointer/CurrentSetpointValues[0]
//     Term 25 (AT2002-0250)/CC Outputs/Current setpoint value Ch.10 <-> Data Pointer/CurrentSetpointValues[9]
//     Term 25 (AT2002-0250)/CC Outputs/Current setpoint value Ch.11 <-> Data Pointer/CurrentSetpointValues[10]
//     Term 25 (AT2002-0250)/CC Outputs/Current setpoint value Ch.12 <-> Data Pointer/CurrentSetpointValues[11]
//     Term 25 (AT2002-0250)/CC Outputs/Current setpoint value Ch.13 <-> Data Pointer/CurrentSetpointValues[12]
//     Term 25 (AT2002-0250)/CC Outputs/Current setpoint value Ch.14 <-> Data Pointer/CurrentSetpointValues[13]
//     Term 25 (AT2002-0250)/CC Outputs/Current setpoint value Ch.15 <-> Data Pointer/CurrentSetpointValues[14]
//     Term 25 (AT2002-0250)/CC Outputs/Current setpoint value Ch.2 <-> Data Pointer/CurrentSetpointValues[1]
//     Term 25 (AT2002-0250)/CC Outputs/Current setpoint value Ch.3 <-> Data Pointer/CurrentSetpointValues[2]
//     Term 25 (AT2002-0250)/CC Outputs/Current setpoint value Ch.4 <-> Data Pointer/CurrentSetpointValues[3]
//     Term 25 (AT2002-0250)/CC Outputs/Current setpoint value Ch.5 <-> Data Pointer/CurrentSetpointValues[4]
//     Term 25 (AT2002-0250)/CC Outputs/Current setpoint value Ch.6 <-> Data Pointer/CurrentSetpointValues[5]
//     Term 25 (AT2002-0250)/CC Outputs/Current setpoint value Ch.7 <-> Data Pointer/CurrentSetpointValues[6]
//     Term 25 (AT2002-0250)/CC Outputs/Current setpoint value Ch.8 <-> Data Pointer/CurrentSetpointValues[7]
//     Term 25 (AT2002-0250)/CC Outputs/Current setpoint value Ch.9 <-> Data Pointer/CurrentSetpointValues[8]
//     Term 25 (AT2002-0250)/Term 26 (AT2002-5250)/FB Inputs/Value Channel 01 <-> Data Pointer/RawPositionValues[0]
//     Term 25 (AT2002-0250)/Term 26 (AT2002-5250)/FB Inputs/Value Channel 02 <-> Data Pointer/RawPositionValues[1]
//     Term 25 (AT2002-0250)/Term 26 (AT2002-5250)/FB Inputs/Value Channel 03 <-> Data Pointer/RawPositionValues[2]
//     Term 25 (AT2002-0250)/Term 26 (AT2002-5250)/FB Inputs/Value Channel 04 <-> Data Pointer/RawPositionValues[3]
//     Term 25 (AT2002-0250)/Term 26 (AT2002-5250)/FB Inputs/Value Channel 05 <-> Data Pointer/RawPositionValues[4]
//     Term 25 (AT2002-0250)/Term 26 (AT2002-5250)/FB Inputs/Value Channel 06 <-> Data Pointer/RawPositionValues[5]
//     Term 25 (AT2002-0250)/Term 26 (AT2002-5250)/FB Inputs/Value Channel 07 <-> Data Pointer/RawPositionValues[6]
//     Term 25 (AT2002-0250)/Term 26 (AT2002-5250)/FB Inputs/Value Channel 08 <-> Data Pointer/RawPositionValues[7]
//     Term 25 (AT2002-0250)/Term 26 (AT2002-5250)/FB Inputs/Value Channel 09 <-> Data Pointer/RawPositionValues[8]
//     Term 25 (AT2002-0250)/Term 26 (AT2002-5250)/FB Inputs/Value Channel 10 <-> Data Pointer/RawPositionValues[9]
//     Term 25 (AT2002-0250)/Term 26 (AT2002-5250)/FB Inputs/Value Channel 11 <-> Data Pointer/RawPositionValues[10]
//     Term 25 (AT2002-0250)/Term 26 (AT2002-5250)/FB Inputs/Value Channel 12 <-> Data Pointer/RawPositionValues[11]
//     Term 25 (AT2002-0250)/Term 26 (AT2002-5250)/FB Inputs/Value Channel 13 <-> Data Pointer/RawPositionValues[12]
//     Term 25 (AT2002-0250)/Term 26 (AT2002-5250)/FB Inputs/Value Channel 14 <-> Data Pointer/RawPositionValues[13]
//     Term 25 (AT2002-0250)/Term 26 (AT2002-5250)/FB Inputs/Value Channel 15 <-> Data Pointer/RawPositionValues[14]
//     Term 25 (AT2002-0250)/Term 26 (AT2002-5250)/FB Inputs/Value Channel 16 <-> Data Pointer/RawPositionValues[15]
//     Term 25 (AT2002-0250)/Term 26 (AT2002-5250)/FB Inputs/Value Channel 17 <-> Data Pointer/RawPositionValues[16]
//     Term 25 (AT2002-0250)/Term 26 (AT2002-5250)/FB Inputs/Value Channel 18 <-> Data Pointer/RawPositionValues[17]
//     Term 25 (AT2002-0250)/Term 26 (AT2002-5250)/FB Inputs/Value Channel 19 <-> Data Pointer/RawPositionValues[18]
//     Term 25 (AT2002-0250)/Term 26 (AT2002-5250)/FB Inputs/Value Channel 20 <-> Data Pointer/RawPositionValues[19]
//     Term 25 (AT2002-0250)/Term 26 (AT2002-5250)/FB Inputs/Value Channel 21 <-> Data Pointer/RawPositionValues[20]
//     Term 25 (AT2002-0250)/Term 26 (AT2002-5250)/FB Inputs/Value Channel 22 <-> Data Pointer/RawPositionValues[21]
//     Term 25 (AT2002-0250)/Term 26 (AT2002-5250)/FB Inputs/Value Channel 23 <-> Data Pointer/RawPositionValues[22]
//     Term 25 (AT2002-0250)/Term 26 (AT2002-5250)/FB Inputs/Value Channel 24 <-> Data Pointer/RawPositionValues[23]
//     Term 25 (AT2002-0250)/Term 26 (AT2002-5250)/FB Inputs/Value Channel 25 <-> Data Pointer/RawPositionValues[24]
//     Term 25 (AT2002-0250)/Term 26 (AT2002-5250)/FB Inputs/Value Channel 26 <-> Data Pointer/RawPositionValues[25]
//     Term 25 (AT2002-0250)/Term 26 (AT2002-5250)/FB Inputs/Value Channel 27 <-> Data Pointer/RawPositionValues[26]
//     Term 25 (AT2002-0250)/Term 26 (AT2002-5250)/FB Inputs/Value Channel 28 <-> Data Pointer/RawPositionValues[27]
//     Term 25 (AT2002-0250)/Term 26 (AT2002-5250)/FB Inputs/Value Channel 29 <-> Data Pointer/RawPositionValues[28]
//     Term 25 (AT2002-0250)/Term 26 (AT2002-5250)/FB Inputs/Value Channel 30 <-> Data Pointer/RawPositionValues[29]
//     Term 25 (AT2002-0250)/Term 26 (AT2002-5250)/FB Inputs/Value Channel 31 <-> Data Pointer/RawPositionValues[30]
//     Term 25 (AT2002-0250)/Term 26 (AT2002-5250)/FB Inputs/Value Channel 32 <-> Data Pointer/RawPositionValues[31]
//   Device 22 <-> TcCOM Objects/XTS ProcessingUnit 1/Part 1/Module 21
//     Term 27 (AT2200-0500)/CC Inputs/Current actual value Ch.1 <-> Data Pointer/CurrentActualValues[0]
//     Term 27 (AT2200-0500)/CC Inputs/Current actual value Ch.10 <-> Data Pointer/CurrentActualValues[9]
//     Term 27 (AT2200-0500)/CC Inputs/Current actual value Ch.11 <-> Data Pointer/CurrentActualValues[10]
//     Term 27 (AT2200-0500)/CC Inputs/Current actual value Ch.12 <-> Data Pointer/CurrentActualValues[11]
//     Term 27 (AT2200-0500)/CC Inputs/Current actual value Ch.13 <-> Data Pointer/CurrentActualValues[12]
//     Term 27 (AT2200-0500)/CC Inputs/Current actual value Ch.14 <-> Data Pointer/CurrentActualValues[13]
//     Term 27 (AT2200-0500)/CC Inputs/Current actual value Ch.15 <-> Data Pointer/CurrentActualValues[14]
//     Term 27 (AT2200-0500)/CC Inputs/Current actual value Ch.16 <-> Data Pointer/CurrentActualValues[15]
//     Term 27 (AT2200-0500)/CC Inputs/Current actual value Ch.17 <-> Data Pointer/CurrentActualValues[16]
//     Term 27 (AT2200-0500)/CC Inputs/Current actual value Ch.18 <-> Data Pointer/CurrentActualValues[17]
//     Term 27 (AT2200-0500)/CC Inputs/Current actual value Ch.19 <-> Data Pointer/CurrentActualValues[18]
//     Term 27 (AT2200-0500)/CC Inputs/Current actual value Ch.2 <-> Data Pointer/CurrentActualValues[1]
//     Term 27 (AT2200-0500)/CC Inputs/Current actual value Ch.20 <-> Data Pointer/CurrentActualValues[19]
//     Term 27 (AT2200-0500)/CC Inputs/Current actual value Ch.21 <-> Data Pointer/CurrentActualValues[20]
//     Term 27 (AT2200-0500)/CC Inputs/Current actual value Ch.22 <-> Data Pointer/CurrentActualValues[21]
//     Term 27 (AT2200-0500)/CC Inputs/Current actual value Ch.23 <-> Data Pointer/CurrentActualValues[22]
//     Term 27 (AT2200-0500)/CC Inputs/Current actual value Ch.24 <-> Data Pointer/CurrentActualValues[23]
//     Term 27 (AT2200-0500)/CC Inputs/Current actual value Ch.25 <-> Data Pointer/CurrentActualValues[24]
//     Term 27 (AT2200-0500)/CC Inputs/Current actual value Ch.26 <-> Data Pointer/CurrentActualValues[25]
//     Term 27 (AT2200-0500)/CC Inputs/Current actual value Ch.27 <-> Data Pointer/CurrentActualValues[26]
//     Term 27 (AT2200-0500)/CC Inputs/Current actual value Ch.28 <-> Data Pointer/CurrentActualValues[27]
//     Term 27 (AT2200-0500)/CC Inputs/Current actual value Ch.29 <-> Data Pointer/CurrentActualValues[28]
//     Term 27 (AT2200-0500)/CC Inputs/Current actual value Ch.3 <-> Data Pointer/CurrentActualValues[2]
//     Term 27 (AT2200-0500)/CC Inputs/Current actual value Ch.30 <-> Data Pointer/CurrentActualValues[29]
//     Term 27 (AT2200-0500)/CC Inputs/Current actual value Ch.4 <-> Data Pointer/CurrentActualValues[3]
//     Term 27 (AT2200-0500)/CC Inputs/Current actual value Ch.5 <-> Data Pointer/CurrentActualValues[4]
//     Term 27 (AT2200-0500)/CC Inputs/Current actual value Ch.6 <-> Data Pointer/CurrentActualValues[5]
//     Term 27 (AT2200-0500)/CC Inputs/Current actual value Ch.7 <-> Data Pointer/CurrentActualValues[6]
//     Term 27 (AT2200-0500)/CC Inputs/Current actual value Ch.8 <-> Data Pointer/CurrentActualValues[7]
//     Term 27 (AT2200-0500)/CC Inputs/Current actual value Ch.9 <-> Data Pointer/CurrentActualValues[8]
//     Term 27 (AT2200-0500)/CC Inputs/Status <-> Data Pointer/Status
//     Term 27 (AT2200-0500)/CC Outputs/Control <-> Data Pointer/Control
//     Term 27 (AT2200-0500)/CC Outputs/Current setpoint value Ch.1 <-> Data Pointer/CurrentSetpointValues[0]
//     Term 27 (AT2200-0500)/CC Outputs/Current setpoint value Ch.10 <-> Data Pointer/CurrentSetpointValues[9]
//     Term 27 (AT2200-0500)/CC Outputs/Current setpoint value Ch.11 <-> Data Pointer/CurrentSetpointValues[10]
//     Term 27 (AT2200-0500)/CC Outputs/Current setpoint value Ch.12 <-> Data Pointer/CurrentSetpointValues[11]
//     Term 27 (AT2200-0500)/CC Outputs/Current setpoint value Ch.13 <-> Data Pointer/CurrentSetpointValues[12]
//     Term 27 (AT2200-0500)/CC Outputs/Current setpoint value Ch.14 <-> Data Pointer/CurrentSetpointValues[13]
//     Term 27 (AT2200-0500)/CC Outputs/Current setpoint value Ch.15 <-> Data Pointer/CurrentSetpointValues[14]
//     Term 27 (AT2200-0500)/CC Outputs/Current setpoint value Ch.16 <-> Data Pointer/CurrentSetpointValues[15]
//     Term 27 (AT2200-0500)/CC Outputs/Current setpoint value Ch.17 <-> Data Pointer/CurrentSetpointValues[16]
//     Term 27 (AT2200-0500)/CC Outputs/Current setpoint value Ch.18 <-> Data Pointer/CurrentSetpointValues[17]
//     Term 27 (AT2200-0500)/CC Outputs/Current setpoint value Ch.19 <-> Data Pointer/CurrentSetpointValues[18]
//     Term 27 (AT2200-0500)/CC Outputs/Current setpoint value Ch.2 <-> Data Pointer/CurrentSetpointValues[1]
//     Term 27 (AT2200-0500)/CC Outputs/Current setpoint value Ch.20 <-> Data Pointer/CurrentSetpointValues[19]
//     Term 27 (AT2200-0500)/CC Outputs/Current setpoint value Ch.21 <-> Data Pointer/CurrentSetpointValues[20]
//     Term 27 (AT2200-0500)/CC Outputs/Current setpoint value Ch.22 <-> Data Pointer/CurrentSetpointValues[21]
//     Term 27 (AT2200-0500)/CC Outputs/Current setpoint value Ch.23 <-> Data Pointer/CurrentSetpointValues[22]
//     Term 27 (AT2200-0500)/CC Outputs/Current setpoint value Ch.24 <-> Data Pointer/CurrentSetpointValues[23]
//     Term 27 (AT2200-0500)/CC Outputs/Current setpoint value Ch.25 <-> Data Pointer/CurrentSetpointValues[24]
//     Term 27 (AT2200-0500)/CC Outputs/Current setpoint value Ch.26 <-> Data Pointer/CurrentSetpointValues[25]
//     Term 27 (AT2200-0500)/CC Outputs/Current setpoint value Ch.27 <-> Data Pointer/CurrentSetpointValues[26]
//     Term 27 (AT2200-0500)/CC Outputs/Current setpoint value Ch.28 <-> Data Pointer/CurrentSetpointValues[27]
//     Term 27 (AT2200-0500)/CC Outputs/Current setpoint value Ch.29 <-> Data Pointer/CurrentSetpointValues[28]
//     Term 27 (AT2200-0500)/CC Outputs/Current setpoint value Ch.3 <-> Data Pointer/CurrentSetpointValues[2]
//     Term 27 (AT2200-0500)/CC Outputs/Current setpoint value Ch.30 <-> Data Pointer/CurrentSetpointValues[29]
//     Term 27 (AT2200-0500)/CC Outputs/Current setpoint value Ch.4 <-> Data Pointer/CurrentSetpointValues[3]
//     Term 27 (AT2200-0500)/CC Outputs/Current setpoint value Ch.5 <-> Data Pointer/CurrentSetpointValues[4]
//     Term 27 (AT2200-0500)/CC Outputs/Current setpoint value Ch.6 <-> Data Pointer/CurrentSetpointValues[5]
//     Term 27 (AT2200-0500)/CC Outputs/Current setpoint value Ch.7 <-> Data Pointer/CurrentSetpointValues[6]
//     Term 27 (AT2200-0500)/CC Outputs/Current setpoint value Ch.8 <-> Data Pointer/CurrentSetpointValues[7]
//     Term 27 (AT2200-0500)/CC Outputs/Current setpoint value Ch.9 <-> Data Pointer/CurrentSetpointValues[8]
//     Term 27 (AT2200-0500)/LFB Inputs/BinaryData <-> Data Pointer/HallSensorValues
//   Device 22 <-> TcCOM Objects/XTS ProcessingUnit 1/Part 1/Module 22
//     Term 28 (AT2200-0500)/CC Inputs/Current actual value Ch.1 <-> Data Pointer/CurrentActualValues[0]
//     Term 28 (AT2200-0500)/CC Inputs/Current actual value Ch.10 <-> Data Pointer/CurrentActualValues[9]
//     Term 28 (AT2200-0500)/CC Inputs/Current actual value Ch.11 <-> Data Pointer/CurrentActualValues[10]
//     Term 28 (AT2200-0500)/CC Inputs/Current actual value Ch.12 <-> Data Pointer/CurrentActualValues[11]
//     Term 28 (AT2200-0500)/CC Inputs/Current actual value Ch.13 <-> Data Pointer/CurrentActualValues[12]
//     Term 28 (AT2200-0500)/CC Inputs/Current actual value Ch.14 <-> Data Pointer/CurrentActualValues[13]
//     Term 28 (AT2200-0500)/CC Inputs/Current actual value Ch.15 <-> Data Pointer/CurrentActualValues[14]
//     Term 28 (AT2200-0500)/CC Inputs/Current actual value Ch.16 <-> Data Pointer/CurrentActualValues[15]
//     Term 28 (AT2200-0500)/CC Inputs/Current actual value Ch.17 <-> Data Pointer/CurrentActualValues[16]
//     Term 28 (AT2200-0500)/CC Inputs/Current actual value Ch.18 <-> Data Pointer/CurrentActualValues[17]
//     Term 28 (AT2200-0500)/CC Inputs/Current actual value Ch.19 <-> Data Pointer/CurrentActualValues[18]
//     Term 28 (AT2200-0500)/CC Inputs/Current actual value Ch.2 <-> Data Pointer/CurrentActualValues[1]
//     Term 28 (AT2200-0500)/CC Inputs/Current actual value Ch.20 <-> Data Pointer/CurrentActualValues[19]
//     Term 28 (AT2200-0500)/CC Inputs/Current actual value Ch.21 <-> Data Pointer/CurrentActualValues[20]
//     Term 28 (AT2200-0500)/CC Inputs/Current actual value Ch.22 <-> Data Pointer/CurrentActualValues[21]
//     Term 28 (AT2200-0500)/CC Inputs/Current actual value Ch.23 <-> Data Pointer/CurrentActualValues[22]
//     Term 28 (AT2200-0500)/CC Inputs/Current actual value Ch.24 <-> Data Pointer/CurrentActualValues[23]
//     Term 28 (AT2200-0500)/CC Inputs/Current actual value Ch.25 <-> Data Pointer/CurrentActualValues[24]
//     Term 28 (AT2200-0500)/CC Inputs/Current actual value Ch.26 <-> Data Pointer/CurrentActualValues[25]
//     Term 28 (AT2200-0500)/CC Inputs/Current actual value Ch.27 <-> Data Pointer/CurrentActualValues[26]
//     Term 28 (AT2200-0500)/CC Inputs/Current actual value Ch.28 <-> Data Pointer/CurrentActualValues[27]
//     Term 28 (AT2200-0500)/CC Inputs/Current actual value Ch.29 <-> Data Pointer/CurrentActualValues[28]
//     Term 28 (AT2200-0500)/CC Inputs/Current actual value Ch.3 <-> Data Pointer/CurrentActualValues[2]
//     Term 28 (AT2200-0500)/CC Inputs/Current actual value Ch.30 <-> Data Pointer/CurrentActualValues[29]
//     Term 28 (AT2200-0500)/CC Inputs/Current actual value Ch.4 <-> Data Pointer/CurrentActualValues[3]
//     Term 28 (AT2200-0500)/CC Inputs/Current actual value Ch.5 <-> Data Pointer/CurrentActualValues[4]
//     Term 28 (AT2200-0500)/CC Inputs/Current actual value Ch.6 <-> Data Pointer/CurrentActualValues[5]
//     Term 28 (AT2200-0500)/CC Inputs/Current actual value Ch.7 <-> Data Pointer/CurrentActualValues[6]
//     Term 28 (AT2200-0500)/CC Inputs/Current actual value Ch.8 <-> Data Pointer/CurrentActualValues[7]
//     Term 28 (AT2200-0500)/CC Inputs/Current actual value Ch.9 <-> Data Pointer/CurrentActualValues[8]
//     Term 28 (AT2200-0500)/CC Inputs/Status <-> Data Pointer/Status
//     Term 28 (AT2200-0500)/CC Outputs/Control <-> Data Pointer/Control
//     Term 28 (AT2200-0500)/CC Outputs/Current setpoint value Ch.1 <-> Data Pointer/CurrentSetpointValues[0]
//     Term 28 (AT2200-0500)/CC Outputs/Current setpoint value Ch.10 <-> Data Pointer/CurrentSetpointValues[9]
//     Term 28 (AT2200-0500)/CC Outputs/Current setpoint value Ch.11 <-> Data Pointer/CurrentSetpointValues[10]
//     Term 28 (AT2200-0500)/CC Outputs/Current setpoint value Ch.12 <-> Data Pointer/CurrentSetpointValues[11]
//     Term 28 (AT2200-0500)/CC Outputs/Current setpoint value Ch.13 <-> Data Pointer/CurrentSetpointValues[12]
//     Term 28 (AT2200-0500)/CC Outputs/Current setpoint value Ch.14 <-> Data Pointer/CurrentSetpointValues[13]
//     Term 28 (AT2200-0500)/CC Outputs/Current setpoint value Ch.15 <-> Data Pointer/CurrentSetpointValues[14]
//     Term 28 (AT2200-0500)/CC Outputs/Current setpoint value Ch.16 <-> Data Pointer/CurrentSetpointValues[15]
//     Term 28 (AT2200-0500)/CC Outputs/Current setpoint value Ch.17 <-> Data Pointer/CurrentSetpointValues[16]
//     Term 28 (AT2200-0500)/CC Outputs/Current setpoint value Ch.18 <-> Data Pointer/CurrentSetpointValues[17]
//     Term 28 (AT2200-0500)/CC Outputs/Current setpoint value Ch.19 <-> Data Pointer/CurrentSetpointValues[18]
//     Term 28 (AT2200-0500)/CC Outputs/Current setpoint value Ch.2 <-> Data Pointer/CurrentSetpointValues[1]
//     Term 28 (AT2200-0500)/CC Outputs/Current setpoint value Ch.20 <-> Data Pointer/CurrentSetpointValues[19]
//     Term 28 (AT2200-0500)/CC Outputs/Current setpoint value Ch.21 <-> Data Pointer/CurrentSetpointValues[20]
//     Term 28 (AT2200-0500)/CC Outputs/Current setpoint value Ch.22 <-> Data Pointer/CurrentSetpointValues[21]
//     Term 28 (AT2200-0500)/CC Outputs/Current setpoint value Ch.23 <-> Data Pointer/CurrentSetpointValues[22]
//     Term 28 (AT2200-0500)/CC Outputs/Current setpoint value Ch.24 <-> Data Pointer/CurrentSetpointValues[23]
//     Term 28 (AT2200-0500)/CC Outputs/Current setpoint value Ch.25 <-> Data Pointer/CurrentSetpointValues[24]
//     Term 28 (AT2200-0500)/CC Outputs/Current setpoint value Ch.26 <-> Data Pointer/CurrentSetpointValues[25]
//     Term 28 (AT2200-0500)/CC Outputs/Current setpoint value Ch.27 <-> Data Pointer/CurrentSetpointValues[26]
//     Term 28 (AT2200-0500)/CC Outputs/Current setpoint value Ch.28 <-> Data Pointer/CurrentSetpointValues[27]
//     Term 28 (AT2200-0500)/CC Outputs/Current setpoint value Ch.29 <-> Data Pointer/CurrentSetpointValues[28]
//     Term 28 (AT2200-0500)/CC Outputs/Current setpoint value Ch.3 <-> Data Pointer/CurrentSetpointValues[2]
//     Term 28 (AT2200-0500)/CC Outputs/Current setpoint value Ch.30 <-> Data Pointer/CurrentSetpointValues[29]
//     Term 28 (AT2200-0500)/CC Outputs/Current setpoint value Ch.4 <-> Data Pointer/CurrentSetpointValues[3]
//     Term 28 (AT2200-0500)/CC Outputs/Current setpoint value Ch.5 <-> Data Pointer/CurrentSetpointValues[4]
//     Term 28 (AT2200-0500)/CC Outputs/Current setpoint value Ch.6 <-> Data Pointer/CurrentSetpointValues[5]
//     Term 28 (AT2200-0500)/CC Outputs/Current setpoint value Ch.7 <-> Data Pointer/CurrentSetpointValues[6]
//     Term 28 (AT2200-0500)/CC Outputs/Current setpoint value Ch.8 <-> Data Pointer/CurrentSetpointValues[7]
//     Term 28 (AT2200-0500)/CC Outputs/Current setpoint value Ch.9 <-> Data Pointer/CurrentSetpointValues[8]
//     Term 28 (AT2200-0500)/LFB Inputs/BinaryData <-> Data Pointer/HallSensorValues
//   Device 23 <-> TcCOM Objects/XTS ProcessingUnit 1/Part 1/Module 23
//     Term 29 (AT2202-0500)/CC Inputs/Current actual value Ch.1 <-> Data Pointer/CurrentActualValues[0]
//     Term 29 (AT2202-0500)/CC Inputs/Current actual value Ch.10 <-> Data Pointer/CurrentActualValues[9]
//     Term 29 (AT2202-0500)/CC Inputs/Current actual value Ch.11 <-> Data Pointer/CurrentActualValues[10]
//     Term 29 (AT2202-0500)/CC Inputs/Current actual value Ch.12 <-> Data Pointer/CurrentActualValues[11]
//     Term 29 (AT2202-0500)/CC Inputs/Current actual value Ch.13 <-> Data Pointer/CurrentActualValues[12]
//     Term 29 (AT2202-0500)/CC Inputs/Current actual value Ch.14 <-> Data Pointer/CurrentActualValues[13]
//     Term 29 (AT2202-0500)/CC Inputs/Current actual value Ch.15 <-> Data Pointer/CurrentActualValues[14]
//     Term 29 (AT2202-0500)/CC Inputs/Current actual value Ch.16 <-> Data Pointer/CurrentActualValues[15]
//     Term 29 (AT2202-0500)/CC Inputs/Current actual value Ch.17 <-> Data Pointer/CurrentActualValues[16]
//     Term 29 (AT2202-0500)/CC Inputs/Current actual value Ch.18 <-> Data Pointer/CurrentActualValues[17]
//     Term 29 (AT2202-0500)/CC Inputs/Current actual value Ch.19 <-> Data Pointer/CurrentActualValues[18]
//     Term 29 (AT2202-0500)/CC Inputs/Current actual value Ch.2 <-> Data Pointer/CurrentActualValues[1]
//     Term 29 (AT2202-0500)/CC Inputs/Current actual value Ch.20 <-> Data Pointer/CurrentActualValues[19]
//     Term 29 (AT2202-0500)/CC Inputs/Current actual value Ch.21 <-> Data Pointer/CurrentActualValues[20]
//     Term 29 (AT2202-0500)/CC Inputs/Current actual value Ch.22 <-> Data Pointer/CurrentActualValues[21]
//     Term 29 (AT2202-0500)/CC Inputs/Current actual value Ch.23 <-> Data Pointer/CurrentActualValues[22]
//     Term 29 (AT2202-0500)/CC Inputs/Current actual value Ch.24 <-> Data Pointer/CurrentActualValues[23]
//     Term 29 (AT2202-0500)/CC Inputs/Current actual value Ch.25 <-> Data Pointer/CurrentActualValues[24]
//     Term 29 (AT2202-0500)/CC Inputs/Current actual value Ch.26 <-> Data Pointer/CurrentActualValues[25]
//     Term 29 (AT2202-0500)/CC Inputs/Current actual value Ch.27 <-> Data Pointer/CurrentActualValues[26]
//     Term 29 (AT2202-0500)/CC Inputs/Current actual value Ch.28 <-> Data Pointer/CurrentActualValues[27]
//     Term 29 (AT2202-0500)/CC Inputs/Current actual value Ch.29 <-> Data Pointer/CurrentActualValues[28]
//     Term 29 (AT2202-0500)/CC Inputs/Current actual value Ch.3 <-> Data Pointer/CurrentActualValues[2]
//     Term 29 (AT2202-0500)/CC Inputs/Current actual value Ch.30 <-> Data Pointer/CurrentActualValues[29]
//     Term 29 (AT2202-0500)/CC Inputs/Current actual value Ch.4 <-> Data Pointer/CurrentActualValues[3]
//     Term 29 (AT2202-0500)/CC Inputs/Current actual value Ch.5 <-> Data Pointer/CurrentActualValues[4]
//     Term 29 (AT2202-0500)/CC Inputs/Current actual value Ch.6 <-> Data Pointer/CurrentActualValues[5]
//     Term 29 (AT2202-0500)/CC Inputs/Current actual value Ch.7 <-> Data Pointer/CurrentActualValues[6]
//     Term 29 (AT2202-0500)/CC Inputs/Current actual value Ch.8 <-> Data Pointer/CurrentActualValues[7]
//     Term 29 (AT2202-0500)/CC Inputs/Current actual value Ch.9 <-> Data Pointer/CurrentActualValues[8]
//     Term 29 (AT2202-0500)/CC Inputs/Status <-> Data Pointer/Status
//     Term 29 (AT2202-0500)/CC Outputs/Control <-> Data Pointer/Control
//     Term 29 (AT2202-0500)/CC Outputs/Current setpoint value Ch.1 <-> Data Pointer/CurrentSetpointValues[0]
//     Term 29 (AT2202-0500)/CC Outputs/Current setpoint value Ch.10 <-> Data Pointer/CurrentSetpointValues[9]
//     Term 29 (AT2202-0500)/CC Outputs/Current setpoint value Ch.11 <-> Data Pointer/CurrentSetpointValues[10]
//     Term 29 (AT2202-0500)/CC Outputs/Current setpoint value Ch.12 <-> Data Pointer/CurrentSetpointValues[11]
//     Term 29 (AT2202-0500)/CC Outputs/Current setpoint value Ch.13 <-> Data Pointer/CurrentSetpointValues[12]
//     Term 29 (AT2202-0500)/CC Outputs/Current setpoint value Ch.14 <-> Data Pointer/CurrentSetpointValues[13]
//     Term 29 (AT2202-0500)/CC Outputs/Current setpoint value Ch.15 <-> Data Pointer/CurrentSetpointValues[14]
//     Term 29 (AT2202-0500)/CC Outputs/Current setpoint value Ch.16 <-> Data Pointer/CurrentSetpointValues[15]
//     Term 29 (AT2202-0500)/CC Outputs/Current setpoint value Ch.17 <-> Data Pointer/CurrentSetpointValues[16]
//     Term 29 (AT2202-0500)/CC Outputs/Current setpoint value Ch.18 <-> Data Pointer/CurrentSetpointValues[17]
//     Term 29 (AT2202-0500)/CC Outputs/Current setpoint value Ch.19 <-> Data Pointer/CurrentSetpointValues[18]
//     Term 29 (AT2202-0500)/CC Outputs/Current setpoint value Ch.2 <-> Data Pointer/CurrentSetpointValues[1]
//     Term 29 (AT2202-0500)/CC Outputs/Current setpoint value Ch.20 <-> Data Pointer/CurrentSetpointValues[19]
//     Term 29 (AT2202-0500)/CC Outputs/Current setpoint value Ch.21 <-> Data Pointer/CurrentSetpointValues[20]
//     Term 29 (AT2202-0500)/CC Outputs/Current setpoint value Ch.22 <-> Data Pointer/CurrentSetpointValues[21]
//     Term 29 (AT2202-0500)/CC Outputs/Current setpoint value Ch.23 <-> Data Pointer/CurrentSetpointValues[22]
//     Term 29 (AT2202-0500)/CC Outputs/Current setpoint value Ch.24 <-> Data Pointer/CurrentSetpointValues[23]
//     Term 29 (AT2202-0500)/CC Outputs/Current setpoint value Ch.25 <-> Data Pointer/CurrentSetpointValues[24]
//     Term 29 (AT2202-0500)/CC Outputs/Current setpoint value Ch.26 <-> Data Pointer/CurrentSetpointValues[25]
//     Term 29 (AT2202-0500)/CC Outputs/Current setpoint value Ch.27 <-> Data Pointer/CurrentSetpointValues[26]
//     Term 29 (AT2202-0500)/CC Outputs/Current setpoint value Ch.28 <-> Data Pointer/CurrentSetpointValues[27]
//     Term 29 (AT2202-0500)/CC Outputs/Current setpoint value Ch.29 <-> Data Pointer/CurrentSetpointValues[28]
//     Term 29 (AT2202-0500)/CC Outputs/Current setpoint value Ch.3 <-> Data Pointer/CurrentSetpointValues[2]
//     Term 29 (AT2202-0500)/CC Outputs/Current setpoint value Ch.30 <-> Data Pointer/CurrentSetpointValues[29]
//     Term 29 (AT2202-0500)/CC Outputs/Current setpoint value Ch.4 <-> Data Pointer/CurrentSetpointValues[3]
//     Term 29 (AT2202-0500)/CC Outputs/Current setpoint value Ch.5 <-> Data Pointer/CurrentSetpointValues[4]
//     Term 29 (AT2202-0500)/CC Outputs/Current setpoint value Ch.6 <-> Data Pointer/CurrentSetpointValues[5]
//     Term 29 (AT2202-0500)/CC Outputs/Current setpoint value Ch.7 <-> Data Pointer/CurrentSetpointValues[6]
//     Term 29 (AT2202-0500)/CC Outputs/Current setpoint value Ch.8 <-> Data Pointer/CurrentSetpointValues[7]
//     Term 29 (AT2202-0500)/CC Outputs/Current setpoint value Ch.9 <-> Data Pointer/CurrentSetpointValues[8]
//     Term 29 (AT2202-0500)/LFB Inputs/BinaryData <-> Data Pointer/HallSensorValues
//   Device 23 <-> TcCOM Objects/XTS ProcessingUnit 1/Part 1/Module 24
//     Term 30 (AT2200-0500)/CC Inputs/Current actual value Ch.1 <-> Data Pointer/CurrentActualValues[0]
//     Term 30 (AT2200-0500)/CC Inputs/Current actual value Ch.10 <-> Data Pointer/CurrentActualValues[9]
//     Term 30 (AT2200-0500)/CC Inputs/Current actual value Ch.11 <-> Data Pointer/CurrentActualValues[10]
//     Term 30 (AT2200-0500)/CC Inputs/Current actual value Ch.12 <-> Data Pointer/CurrentActualValues[11]
//     Term 30 (AT2200-0500)/CC Inputs/Current actual value Ch.13 <-> Data Pointer/CurrentActualValues[12]
//     Term 30 (AT2200-0500)/CC Inputs/Current actual value Ch.14 <-> Data Pointer/CurrentActualValues[13]
//     Term 30 (AT2200-0500)/CC Inputs/Current actual value Ch.15 <-> Data Pointer/CurrentActualValues[14]
//     Term 30 (AT2200-0500)/CC Inputs/Current actual value Ch.16 <-> Data Pointer/CurrentActualValues[15]
//     Term 30 (AT2200-0500)/CC Inputs/Current actual value Ch.17 <-> Data Pointer/CurrentActualValues[16]
//     Term 30 (AT2200-0500)/CC Inputs/Current actual value Ch.18 <-> Data Pointer/CurrentActualValues[17]
//     Term 30 (AT2200-0500)/CC Inputs/Current actual value Ch.19 <-> Data Pointer/CurrentActualValues[18]
//     Term 30 (AT2200-0500)/CC Inputs/Current actual value Ch.2 <-> Data Pointer/CurrentActualValues[1]
//     Term 30 (AT2200-0500)/CC Inputs/Current actual value Ch.20 <-> Data Pointer/CurrentActualValues[19]
//     Term 30 (AT2200-0500)/CC Inputs/Current actual value Ch.21 <-> Data Pointer/CurrentActualValues[20]
//     Term 30 (AT2200-0500)/CC Inputs/Current actual value Ch.22 <-> Data Pointer/CurrentActualValues[21]
//     Term 30 (AT2200-0500)/CC Inputs/Current actual value Ch.23 <-> Data Pointer/CurrentActualValues[22]
//     Term 30 (AT2200-0500)/CC Inputs/Current actual value Ch.24 <-> Data Pointer/CurrentActualValues[23]
//     Term 30 (AT2200-0500)/CC Inputs/Current actual value Ch.25 <-> Data Pointer/CurrentActualValues[24]
//     Term 30 (AT2200-0500)/CC Inputs/Current actual value Ch.26 <-> Data Pointer/CurrentActualValues[25]
//     Term 30 (AT2200-0500)/CC Inputs/Current actual value Ch.27 <-> Data Pointer/CurrentActualValues[26]
//     Term 30 (AT2200-0500)/CC Inputs/Current actual value Ch.28 <-> Data Pointer/CurrentActualValues[27]
//     Term 30 (AT2200-0500)/CC Inputs/Current actual value Ch.29 <-> Data Pointer/CurrentActualValues[28]
//     Term 30 (AT2200-0500)/CC Inputs/Current actual value Ch.3 <-> Data Pointer/CurrentActualValues[2]
//     Term 30 (AT2200-0500)/CC Inputs/Current actual value Ch.30 <-> Data Pointer/CurrentActualValues[29]
//     Term 30 (AT2200-0500)/CC Inputs/Current actual value Ch.4 <-> Data Pointer/CurrentActualValues[3]
//     Term 30 (AT2200-0500)/CC Inputs/Current actual value Ch.5 <-> Data Pointer/CurrentActualValues[4]
//     Term 30 (AT2200-0500)/CC Inputs/Current actual value Ch.6 <-> Data Pointer/CurrentActualValues[5]
//     Term 30 (AT2200-0500)/CC Inputs/Current actual value Ch.7 <-> Data Pointer/CurrentActualValues[6]
//     Term 30 (AT2200-0500)/CC Inputs/Current actual value Ch.8 <-> Data Pointer/CurrentActualValues[7]
//     Term 30 (AT2200-0500)/CC Inputs/Current actual value Ch.9 <-> Data Pointer/CurrentActualValues[8]
//     Term 30 (AT2200-0500)/CC Inputs/Status <-> Data Pointer/Status
//     Term 30 (AT2200-0500)/CC Outputs/Control <-> Data Pointer/Control
//     Term 30 (AT2200-0500)/CC Outputs/Current setpoint value Ch.1 <-> Data Pointer/CurrentSetpointValues[0]
//     Term 30 (AT2200-0500)/CC Outputs/Current setpoint value Ch.10 <-> Data Pointer/CurrentSetpointValues[9]
//     Term 30 (AT2200-0500)/CC Outputs/Current setpoint value Ch.11 <-> Data Pointer/CurrentSetpointValues[10]
//     Term 30 (AT2200-0500)/CC Outputs/Current setpoint value Ch.12 <-> Data Pointer/CurrentSetpointValues[11]
//     Term 30 (AT2200-0500)/CC Outputs/Current setpoint value Ch.13 <-> Data Pointer/CurrentSetpointValues[12]
//     Term 30 (AT2200-0500)/CC Outputs/Current setpoint value Ch.14 <-> Data Pointer/CurrentSetpointValues[13]
//     Term 30 (AT2200-0500)/CC Outputs/Current setpoint value Ch.15 <-> Data Pointer/CurrentSetpointValues[14]
//     Term 30 (AT2200-0500)/CC Outputs/Current setpoint value Ch.16 <-> Data Pointer/CurrentSetpointValues[15]
//     Term 30 (AT2200-0500)/CC Outputs/Current setpoint value Ch.17 <-> Data Pointer/CurrentSetpointValues[16]
//     Term 30 (AT2200-0500)/CC Outputs/Current setpoint value Ch.18 <-> Data Pointer/CurrentSetpointValues[17]
//     Term 30 (AT2200-0500)/CC Outputs/Current setpoint value Ch.19 <-> Data Pointer/CurrentSetpointValues[18]
//     Term 30 (AT2200-0500)/CC Outputs/Current setpoint value Ch.2 <-> Data Pointer/CurrentSetpointValues[1]
//     Term 30 (AT2200-0500)/CC Outputs/Current setpoint value Ch.20 <-> Data Pointer/CurrentSetpointValues[19]
//     Term 30 (AT2200-0500)/CC Outputs/Current setpoint value Ch.21 <-> Data Pointer/CurrentSetpointValues[20]
//     Term 30 (AT2200-0500)/CC Outputs/Current setpoint value Ch.22 <-> Data Pointer/CurrentSetpointValues[21]
//     Term 30 (AT2200-0500)/CC Outputs/Current setpoint value Ch.23 <-> Data Pointer/CurrentSetpointValues[22]
//     Term 30 (AT2200-0500)/CC Outputs/Current setpoint value Ch.24 <-> Data Pointer/CurrentSetpointValues[23]
//     Term 30 (AT2200-0500)/CC Outputs/Current setpoint value Ch.25 <-> Data Pointer/CurrentSetpointValues[24]
//     Term 30 (AT2200-0500)/CC Outputs/Current setpoint value Ch.26 <-> Data Pointer/CurrentSetpointValues[25]
//     Term 30 (AT2200-0500)/CC Outputs/Current setpoint value Ch.27 <-> Data Pointer/CurrentSetpointValues[26]
//     Term 30 (AT2200-0500)/CC Outputs/Current setpoint value Ch.28 <-> Data Pointer/CurrentSetpointValues[27]
//     Term 30 (AT2200-0500)/CC Outputs/Current setpoint value Ch.29 <-> Data Pointer/CurrentSetpointValues[28]
//     Term 30 (AT2200-0500)/CC Outputs/Current setpoint value Ch.3 <-> Data Pointer/CurrentSetpointValues[2]
//     Term 30 (AT2200-0500)/CC Outputs/Current setpoint value Ch.30 <-> Data Pointer/CurrentSetpointValues[29]
//     Term 30 (AT2200-0500)/CC Outputs/Current setpoint value Ch.4 <-> Data Pointer/CurrentSetpointValues[3]
//     Term 30 (AT2200-0500)/CC Outputs/Current setpoint value Ch.5 <-> Data Pointer/CurrentSetpointValues[4]
//     Term 30 (AT2200-0500)/CC Outputs/Current setpoint value Ch.6 <-> Data Pointer/CurrentSetpointValues[5]
//     Term 30 (AT2200-0500)/CC Outputs/Current setpoint value Ch.7 <-> Data Pointer/CurrentSetpointValues[6]
//     Term 30 (AT2200-0500)/CC Outputs/Current setpoint value Ch.8 <-> Data Pointer/CurrentSetpointValues[7]
//     Term 30 (AT2200-0500)/CC Outputs/Current setpoint value Ch.9 <-> Data Pointer/CurrentSetpointValues[8]
//     Term 30 (AT2200-0500)/LFB Inputs/BinaryData <-> Data Pointer/HallSensorValues
//   Device 23 <-> TcCOM Objects/XTS ProcessingUnit 1/Part 1/Module 25
//     Term 31 (AT2040-0250)/CC Inputs/Current actual value Ch.1 <-> Data Pointer/CurrentActualValues[0]
//     Term 31 (AT2040-0250)/CC Inputs/Current actual value Ch.10 <-> Data Pointer/CurrentActualValues[9]
//     Term 31 (AT2040-0250)/CC Inputs/Current actual value Ch.11 <-> Data Pointer/CurrentActualValues[10]
//     Term 31 (AT2040-0250)/CC Inputs/Current actual value Ch.12 <-> Data Pointer/CurrentActualValues[11]
//     Term 31 (AT2040-0250)/CC Inputs/Current actual value Ch.13 <-> Data Pointer/CurrentActualValues[12]
//     Term 31 (AT2040-0250)/CC Inputs/Current actual value Ch.14 <-> Data Pointer/CurrentActualValues[13]
//     Term 31 (AT2040-0250)/CC Inputs/Current actual value Ch.15 <-> Data Pointer/CurrentActualValues[14]
//     Term 31 (AT2040-0250)/CC Inputs/Current actual value Ch.2 <-> Data Pointer/CurrentActualValues[1]
//     Term 31 (AT2040-0250)/CC Inputs/Current actual value Ch.3 <-> Data Pointer/CurrentActualValues[2]
//     Term 31 (AT2040-0250)/CC Inputs/Current actual value Ch.4 <-> Data Pointer/CurrentActualValues[3]
//     Term 31 (AT2040-0250)/CC Inputs/Current actual value Ch.5 <-> Data Pointer/CurrentActualValues[4]
//     Term 31 (AT2040-0250)/CC Inputs/Current actual value Ch.6 <-> Data Pointer/CurrentActualValues[5]
//     Term 31 (AT2040-0250)/CC Inputs/Current actual value Ch.7 <-> Data Pointer/CurrentActualValues[6]
//     Term 31 (AT2040-0250)/CC Inputs/Current actual value Ch.8 <-> Data Pointer/CurrentActualValues[7]
//     Term 31 (AT2040-0250)/CC Inputs/Current actual value Ch.9 <-> Data Pointer/CurrentActualValues[8]
//     Term 31 (AT2040-0250)/CC Inputs/Status <-> Data Pointer/Status
//     Term 31 (AT2040-0250)/CC Outputs/Control <-> Data Pointer/Control
//     Term 31 (AT2040-0250)/CC Outputs/Current setpoint value Ch.1 <-> Data Pointer/CurrentSetpointValues[0]
//     Term 31 (AT2040-0250)/CC Outputs/Current setpoint value Ch.10 <-> Data Pointer/CurrentSetpointValues[9]
//     Term 31 (AT2040-0250)/CC Outputs/Current setpoint value Ch.11 <-> Data Pointer/CurrentSetpointValues[10]
//     Term 31 (AT2040-0250)/CC Outputs/Current setpoint value Ch.12 <-> Data Pointer/CurrentSetpointValues[11]
//     Term 31 (AT2040-0250)/CC Outputs/Current setpoint value Ch.13 <-> Data Pointer/CurrentSetpointValues[12]
//     Term 31 (AT2040-0250)/CC Outputs/Current setpoint value Ch.14 <-> Data Pointer/CurrentSetpointValues[13]
//     Term 31 (AT2040-0250)/CC Outputs/Current setpoint value Ch.15 <-> Data Pointer/CurrentSetpointValues[14]
//     Term 31 (AT2040-0250)/CC Outputs/Current setpoint value Ch.2 <-> Data Pointer/CurrentSetpointValues[1]
//     Term 31 (AT2040-0250)/CC Outputs/Current setpoint value Ch.3 <-> Data Pointer/CurrentSetpointValues[2]
//     Term 31 (AT2040-0250)/CC Outputs/Current setpoint value Ch.4 <-> Data Pointer/CurrentSetpointValues[3]
//     Term 31 (AT2040-0250)/CC Outputs/Current setpoint value Ch.5 <-> Data Pointer/CurrentSetpointValues[4]
//     Term 31 (AT2040-0250)/CC Outputs/Current setpoint value Ch.6 <-> Data Pointer/CurrentSetpointValues[5]
//     Term 31 (AT2040-0250)/CC Outputs/Current setpoint value Ch.7 <-> Data Pointer/CurrentSetpointValues[6]
//     Term 31 (AT2040-0250)/CC Outputs/Current setpoint value Ch.8 <-> Data Pointer/CurrentSetpointValues[7]
//     Term 31 (AT2040-0250)/CC Outputs/Current setpoint value Ch.9 <-> Data Pointer/CurrentSetpointValues[8]
//     Term 31 (AT2040-0250)/Term 32 (AT2040-5250)/FB Inputs/Value Channel 01 <-> Data Pointer/RawPositionValues[0]
//     Term 31 (AT2040-0250)/Term 32 (AT2040-5250)/FB Inputs/Value Channel 02 <-> Data Pointer/RawPositionValues[1]
//     Term 31 (AT2040-0250)/Term 32 (AT2040-5250)/FB Inputs/Value Channel 03 <-> Data Pointer/RawPositionValues[2]
//     Term 31 (AT2040-0250)/Term 32 (AT2040-5250)/FB Inputs/Value Channel 04 <-> Data Pointer/RawPositionValues[3]
//     Term 31 (AT2040-0250)/Term 32 (AT2040-5250)/FB Inputs/Value Channel 05 <-> Data Pointer/RawPositionValues[4]
//     Term 31 (AT2040-0250)/Term 32 (AT2040-5250)/FB Inputs/Value Channel 06 <-> Data Pointer/RawPositionValues[5]
//     Term 31 (AT2040-0250)/Term 32 (AT2040-5250)/FB Inputs/Value Channel 07 <-> Data Pointer/RawPositionValues[6]
//     Term 31 (AT2040-0250)/Term 32 (AT2040-5250)/FB Inputs/Value Channel 08 <-> Data Pointer/RawPositionValues[7]
//     Term 31 (AT2040-0250)/Term 32 (AT2040-5250)/FB Inputs/Value Channel 09 <-> Data Pointer/RawPositionValues[8]
//     Term 31 (AT2040-0250)/Term 32 (AT2040-5250)/FB Inputs/Value Channel 10 <-> Data Pointer/RawPositionValues[9]
//     Term 31 (AT2040-0250)/Term 32 (AT2040-5250)/FB Inputs/Value Channel 11 <-> Data Pointer/RawPositionValues[10]
//     Term 31 (AT2040-0250)/Term 32 (AT2040-5250)/FB Inputs/Value Channel 12 <-> Data Pointer/RawPositionValues[11]
//     Term 31 (AT2040-0250)/Term 32 (AT2040-5250)/FB Inputs/Value Channel 13 <-> Data Pointer/RawPositionValues[12]
//     Term 31 (AT2040-0250)/Term 32 (AT2040-5250)/FB Inputs/Value Channel 14 <-> Data Pointer/RawPositionValues[13]
//     Term 31 (AT2040-0250)/Term 32 (AT2040-5250)/FB Inputs/Value Channel 15 <-> Data Pointer/RawPositionValues[14]
//     Term 31 (AT2040-0250)/Term 32 (AT2040-5250)/FB Inputs/Value Channel 16 <-> Data Pointer/RawPositionValues[15]
//     Term 31 (AT2040-0250)/Term 32 (AT2040-5250)/FB Inputs/Value Channel 17 <-> Data Pointer/RawPositionValues[16]
//     Term 31 (AT2040-0250)/Term 32 (AT2040-5250)/FB Inputs/Value Channel 18 <-> Data Pointer/RawPositionValues[17]
//     Term 31 (AT2040-0250)/Term 32 (AT2040-5250)/FB Inputs/Value Channel 19 <-> Data Pointer/RawPositionValues[18]
//     Term 31 (AT2040-0250)/Term 32 (AT2040-5250)/FB Inputs/Value Channel 20 <-> Data Pointer/RawPositionValues[19]
//     Term 31 (AT2040-0250)/Term 32 (AT2040-5250)/FB Inputs/Value Channel 21 <-> Data Pointer/RawPositionValues[20]
//     Term 31 (AT2040-0250)/Term 32 (AT2040-5250)/FB Inputs/Value Channel 22 <-> Data Pointer/RawPositionValues[21]
//     Term 31 (AT2040-0250)/Term 32 (AT2040-5250)/FB Inputs/Value Channel 23 <-> Data Pointer/RawPositionValues[22]
//     Term 31 (AT2040-0250)/Term 32 (AT2040-5250)/FB Inputs/Value Channel 24 <-> Data Pointer/RawPositionValues[23]
//     Term 31 (AT2040-0250)/Term 32 (AT2040-5250)/FB Inputs/Value Channel 25 <-> Data Pointer/RawPositionValues[24]
//     Term 31 (AT2040-0250)/Term 32 (AT2040-5250)/FB Inputs/Value Channel 26 <-> Data Pointer/RawPositionValues[25]
//     Term 31 (AT2040-0250)/Term 32 (AT2040-5250)/FB Inputs/Value Channel 27 <-> Data Pointer/RawPositionValues[26]
//     Term 31 (AT2040-0250)/Term 32 (AT2040-5250)/FB Inputs/Value Channel 28 <-> Data Pointer/RawPositionValues[27]
//     Term 31 (AT2040-0250)/Term 32 (AT2040-5250)/FB Inputs/Value Channel 29 <-> Data Pointer/RawPositionValues[28]
//     Term 31 (AT2040-0250)/Term 32 (AT2040-5250)/FB Inputs/Value Channel 30 <-> Data Pointer/RawPositionValues[29]
//     Term 31 (AT2040-0250)/Term 32 (AT2040-5250)/FB Inputs/Value Channel 31 <-> Data Pointer/RawPositionValues[30]
//     Term 31 (AT2040-0250)/Term 32 (AT2040-5250)/FB Inputs/Value Channel 32 <-> Data Pointer/RawPositionValues[31]
//   Device 24 <-> TcCOM Objects/XTS ProcessingUnit 1/Part 1/Module 26
//     Term 33 (AT2042-0250)/CC Inputs/Current actual value Ch.1 <-> Data Pointer/CurrentActualValues[0]
//     Term 33 (AT2042-0250)/CC Inputs/Current actual value Ch.10 <-> Data Pointer/CurrentActualValues[9]
//     Term 33 (AT2042-0250)/CC Inputs/Current actual value Ch.11 <-> Data Pointer/CurrentActualValues[10]
//     Term 33 (AT2042-0250)/CC Inputs/Current actual value Ch.12 <-> Data Pointer/CurrentActualValues[11]
//     Term 33 (AT2042-0250)/CC Inputs/Current actual value Ch.13 <-> Data Pointer/CurrentActualValues[12]
//     Term 33 (AT2042-0250)/CC Inputs/Current actual value Ch.14 <-> Data Pointer/CurrentActualValues[13]
//     Term 33 (AT2042-0250)/CC Inputs/Current actual value Ch.15 <-> Data Pointer/CurrentActualValues[14]
//     Term 33 (AT2042-0250)/CC Inputs/Current actual value Ch.2 <-> Data Pointer/CurrentActualValues[1]
//     Term 33 (AT2042-0250)/CC Inputs/Current actual value Ch.3 <-> Data Pointer/CurrentActualValues[2]
//     Term 33 (AT2042-0250)/CC Inputs/Current actual value Ch.4 <-> Data Pointer/CurrentActualValues[3]
//     Term 33 (AT2042-0250)/CC Inputs/Current actual value Ch.5 <-> Data Pointer/CurrentActualValues[4]
//     Term 33 (AT2042-0250)/CC Inputs/Current actual value Ch.6 <-> Data Pointer/CurrentActualValues[5]
//     Term 33 (AT2042-0250)/CC Inputs/Current actual value Ch.7 <-> Data Pointer/CurrentActualValues[6]
//     Term 33 (AT2042-0250)/CC Inputs/Current actual value Ch.8 <-> Data Pointer/CurrentActualValues[7]
//     Term 33 (AT2042-0250)/CC Inputs/Current actual value Ch.9 <-> Data Pointer/CurrentActualValues[8]
//     Term 33 (AT2042-0250)/CC Inputs/Status <-> Data Pointer/Status
//     Term 33 (AT2042-0250)/CC Outputs/Control <-> Data Pointer/Control
//     Term 33 (AT2042-0250)/CC Outputs/Current setpoint value Ch.1 <-> Data Pointer/CurrentSetpointValues[0]
//     Term 33 (AT2042-0250)/CC Outputs/Current setpoint value Ch.10 <-> Data Pointer/CurrentSetpointValues[9]
//     Term 33 (AT2042-0250)/CC Outputs/Current setpoint value Ch.11 <-> Data Pointer/CurrentSetpointValues[10]
//     Term 33 (AT2042-0250)/CC Outputs/Current setpoint value Ch.12 <-> Data Pointer/CurrentSetpointValues[11]
//     Term 33 (AT2042-0250)/CC Outputs/Current setpoint value Ch.13 <-> Data Pointer/CurrentSetpointValues[12]
//     Term 33 (AT2042-0250)/CC Outputs/Current setpoint value Ch.14 <-> Data Pointer/CurrentSetpointValues[13]
//     Term 33 (AT2042-0250)/CC Outputs/Current setpoint value Ch.15 <-> Data Pointer/CurrentSetpointValues[14]
//     Term 33 (AT2042-0250)/CC Outputs/Current setpoint value Ch.2 <-> Data Pointer/CurrentSetpointValues[1]
//     Term 33 (AT2042-0250)/CC Outputs/Current setpoint value Ch.3 <-> Data Pointer/CurrentSetpointValues[2]
//     Term 33 (AT2042-0250)/CC Outputs/Current setpoint value Ch.4 <-> Data Pointer/CurrentSetpointValues[3]
//     Term 33 (AT2042-0250)/CC Outputs/Current setpoint value Ch.5 <-> Data Pointer/CurrentSetpointValues[4]
//     Term 33 (AT2042-0250)/CC Outputs/Current setpoint value Ch.6 <-> Data Pointer/CurrentSetpointValues[5]
//     Term 33 (AT2042-0250)/CC Outputs/Current setpoint value Ch.7 <-> Data Pointer/CurrentSetpointValues[6]
//     Term 33 (AT2042-0250)/CC Outputs/Current setpoint value Ch.8 <-> Data Pointer/CurrentSetpointValues[7]
//     Term 33 (AT2042-0250)/CC Outputs/Current setpoint value Ch.9 <-> Data Pointer/CurrentSetpointValues[8]
//     Term 33 (AT2042-0250)/Term 34 (AT2042-5250)/FB Inputs/Value Channel 01 <-> Data Pointer/RawPositionValues[0]
//     Term 33 (AT2042-0250)/Term 34 (AT2042-5250)/FB Inputs/Value Channel 02 <-> Data Pointer/RawPositionValues[1]
//     Term 33 (AT2042-0250)/Term 34 (AT2042-5250)/FB Inputs/Value Channel 03 <-> Data Pointer/RawPositionValues[2]
//     Term 33 (AT2042-0250)/Term 34 (AT2042-5250)/FB Inputs/Value Channel 04 <-> Data Pointer/RawPositionValues[3]
//     Term 33 (AT2042-0250)/Term 34 (AT2042-5250)/FB Inputs/Value Channel 05 <-> Data Pointer/RawPositionValues[4]
//     Term 33 (AT2042-0250)/Term 34 (AT2042-5250)/FB Inputs/Value Channel 06 <-> Data Pointer/RawPositionValues[5]
//     Term 33 (AT2042-0250)/Term 34 (AT2042-5250)/FB Inputs/Value Channel 07 <-> Data Pointer/RawPositionValues[6]
//     Term 33 (AT2042-0250)/Term 34 (AT2042-5250)/FB Inputs/Value Channel 08 <-> Data Pointer/RawPositionValues[7]
//     Term 33 (AT2042-0250)/Term 34 (AT2042-5250)/FB Inputs/Value Channel 09 <-> Data Pointer/RawPositionValues[8]
//     Term 33 (AT2042-0250)/Term 34 (AT2042-5250)/FB Inputs/Value Channel 10 <-> Data Pointer/RawPositionValues[9]
//     Term 33 (AT2042-0250)/Term 34 (AT2042-5250)/FB Inputs/Value Channel 11 <-> Data Pointer/RawPositionValues[10]
//     Term 33 (AT2042-0250)/Term 34 (AT2042-5250)/FB Inputs/Value Channel 12 <-> Data Pointer/RawPositionValues[11]
//     Term 33 (AT2042-0250)/Term 34 (AT2042-5250)/FB Inputs/Value Channel 13 <-> Data Pointer/RawPositionValues[12]
//     Term 33 (AT2042-0250)/Term 34 (AT2042-5250)/FB Inputs/Value Channel 14 <-> Data Pointer/RawPositionValues[13]
//     Term 33 (AT2042-0250)/Term 34 (AT2042-5250)/FB Inputs/Value Channel 15 <-> Data Pointer/RawPositionValues[14]
//     Term 33 (AT2042-0250)/Term 34 (AT2042-5250)/FB Inputs/Value Channel 16 <-> Data Pointer/RawPositionValues[15]
//     Term 33 (AT2042-0250)/Term 34 (AT2042-5250)/FB Inputs/Value Channel 17 <-> Data Pointer/RawPositionValues[16]
//     Term 33 (AT2042-0250)/Term 34 (AT2042-5250)/FB Inputs/Value Channel 18 <-> Data Pointer/RawPositionValues[17]
//     Term 33 (AT2042-0250)/Term 34 (AT2042-5250)/FB Inputs/Value Channel 19 <-> Data Pointer/RawPositionValues[18]
//     Term 33 (AT2042-0250)/Term 34 (AT2042-5250)/FB Inputs/Value Channel 20 <-> Data Pointer/RawPositionValues[19]
//     Term 33 (AT2042-0250)/Term 34 (AT2042-5250)/FB Inputs/Value Channel 21 <-> Data Pointer/RawPositionValues[20]
//     Term 33 (AT2042-0250)/Term 34 (AT2042-5250)/FB Inputs/Value Channel 22 <-> Data Pointer/RawPositionValues[21]
//     Term 33 (AT2042-0250)/Term 34 (AT2042-5250)/FB Inputs/Value Channel 23 <-> Data Pointer/RawPositionValues[22]
//     Term 33 (AT2042-0250)/Term 34 (AT2042-5250)/FB Inputs/Value Channel 24 <-> Data Pointer/RawPositionValues[23]
//     Term 33 (AT2042-0250)/Term 34 (AT2042-5250)/FB Inputs/Value Channel 25 <-> Data Pointer/RawPositionValues[24]
//     Term 33 (AT2042-0250)/Term 34 (AT2042-5250)/FB Inputs/Value Channel 26 <-> Data Pointer/RawPositionValues[25]
//     Term 33 (AT2042-0250)/Term 34 (AT2042-5250)/FB Inputs/Value Channel 27 <-> Data Pointer/RawPositionValues[26]
//     Term 33 (AT2042-0250)/Term 34 (AT2042-5250)/FB Inputs/Value Channel 28 <-> Data Pointer/RawPositionValues[27]
//     Term 33 (AT2042-0250)/Term 34 (AT2042-5250)/FB Inputs/Value Channel 29 <-> Data Pointer/RawPositionValues[28]
//     Term 33 (AT2042-0250)/Term 34 (AT2042-5250)/FB Inputs/Value Channel 30 <-> Data Pointer/RawPositionValues[29]
//     Term 33 (AT2042-0250)/Term 34 (AT2042-5250)/FB Inputs/Value Channel 31 <-> Data Pointer/RawPositionValues[30]
//     Term 33 (AT2042-0250)/Term 34 (AT2042-5250)/FB Inputs/Value Channel 32 <-> Data Pointer/RawPositionValues[31]
//   Device 24 <-> TcCOM Objects/XTS ProcessingUnit 1/Part 1/Module 27
//     Term 35 (AT2200-0500)/CC Inputs/Current actual value Ch.1 <-> Data Pointer/CurrentActualValues[0]
//     Term 35 (AT2200-0500)/CC Inputs/Current actual value Ch.10 <-> Data Pointer/CurrentActualValues[9]
//     Term 35 (AT2200-0500)/CC Inputs/Current actual value Ch.11 <-> Data Pointer/CurrentActualValues[10]
//     Term 35 (AT2200-0500)/CC Inputs/Current actual value Ch.12 <-> Data Pointer/CurrentActualValues[11]
//     Term 35 (AT2200-0500)/CC Inputs/Current actual value Ch.13 <-> Data Pointer/CurrentActualValues[12]
//     Term 35 (AT2200-0500)/CC Inputs/Current actual value Ch.14 <-> Data Pointer/CurrentActualValues[13]
//     Term 35 (AT2200-0500)/CC Inputs/Current actual value Ch.15 <-> Data Pointer/CurrentActualValues[14]
//     Term 35 (AT2200-0500)/CC Inputs/Current actual value Ch.16 <-> Data Pointer/CurrentActualValues[15]
//     Term 35 (AT2200-0500)/CC Inputs/Current actual value Ch.17 <-> Data Pointer/CurrentActualValues[16]
//     Term 35 (AT2200-0500)/CC Inputs/Current actual value Ch.18 <-> Data Pointer/CurrentActualValues[17]
//     Term 35 (AT2200-0500)/CC Inputs/Current actual value Ch.19 <-> Data Pointer/CurrentActualValues[18]
//     Term 35 (AT2200-0500)/CC Inputs/Current actual value Ch.2 <-> Data Pointer/CurrentActualValues[1]
//     Term 35 (AT2200-0500)/CC Inputs/Current actual value Ch.20 <-> Data Pointer/CurrentActualValues[19]
//     Term 35 (AT2200-0500)/CC Inputs/Current actual value Ch.21 <-> Data Pointer/CurrentActualValues[20]
//     Term 35 (AT2200-0500)/CC Inputs/Current actual value Ch.22 <-> Data Pointer/CurrentActualValues[21]
//     Term 35 (AT2200-0500)/CC Inputs/Current actual value Ch.23 <-> Data Pointer/CurrentActualValues[22]
//     Term 35 (AT2200-0500)/CC Inputs/Current actual value Ch.24 <-> Data Pointer/CurrentActualValues[23]
//     Term 35 (AT2200-0500)/CC Inputs/Current actual value Ch.25 <-> Data Pointer/CurrentActualValues[24]
//     Term 35 (AT2200-0500)/CC Inputs/Current actual value Ch.26 <-> Data Pointer/CurrentActualValues[25]
//     Term 35 (AT2200-0500)/CC Inputs/Current actual value Ch.27 <-> Data Pointer/CurrentActualValues[26]
//     Term 35 (AT2200-0500)/CC Inputs/Current actual value Ch.28 <-> Data Pointer/CurrentActualValues[27]
//     Term 35 (AT2200-0500)/CC Inputs/Current actual value Ch.29 <-> Data Pointer/CurrentActualValues[28]
//     Term 35 (AT2200-0500)/CC Inputs/Current actual value Ch.3 <-> Data Pointer/CurrentActualValues[2]
//     Term 35 (AT2200-0500)/CC Inputs/Current actual value Ch.30 <-> Data Pointer/CurrentActualValues[29]
//     Term 35 (AT2200-0500)/CC Inputs/Current actual value Ch.4 <-> Data Pointer/CurrentActualValues[3]
//     Term 35 (AT2200-0500)/CC Inputs/Current actual value Ch.5 <-> Data Pointer/CurrentActualValues[4]
//     Term 35 (AT2200-0500)/CC Inputs/Current actual value Ch.6 <-> Data Pointer/CurrentActualValues[5]
//     Term 35 (AT2200-0500)/CC Inputs/Current actual value Ch.7 <-> Data Pointer/CurrentActualValues[6]
//     Term 35 (AT2200-0500)/CC Inputs/Current actual value Ch.8 <-> Data Pointer/CurrentActualValues[7]
//     Term 35 (AT2200-0500)/CC Inputs/Current actual value Ch.9 <-> Data Pointer/CurrentActualValues[8]
//     Term 35 (AT2200-0500)/CC Inputs/Status <-> Data Pointer/Status
//     Term 35 (AT2200-0500)/CC Outputs/Control <-> Data Pointer/Control
//     Term 35 (AT2200-0500)/CC Outputs/Current setpoint value Ch.1 <-> Data Pointer/CurrentSetpointValues[0]
//     Term 35 (AT2200-0500)/CC Outputs/Current setpoint value Ch.10 <-> Data Pointer/CurrentSetpointValues[9]
//     Term 35 (AT2200-0500)/CC Outputs/Current setpoint value Ch.11 <-> Data Pointer/CurrentSetpointValues[10]
//     Term 35 (AT2200-0500)/CC Outputs/Current setpoint value Ch.12 <-> Data Pointer/CurrentSetpointValues[11]
//     Term 35 (AT2200-0500)/CC Outputs/Current setpoint value Ch.13 <-> Data Pointer/CurrentSetpointValues[12]
//     Term 35 (AT2200-0500)/CC Outputs/Current setpoint value Ch.14 <-> Data Pointer/CurrentSetpointValues[13]
//     Term 35 (AT2200-0500)/CC Outputs/Current setpoint value Ch.15 <-> Data Pointer/CurrentSetpointValues[14]
//     Term 35 (AT2200-0500)/CC Outputs/Current setpoint value Ch.16 <-> Data Pointer/CurrentSetpointValues[15]
//     Term 35 (AT2200-0500)/CC Outputs/Current setpoint value Ch.17 <-> Data Pointer/CurrentSetpointValues[16]
//     Term 35 (AT2200-0500)/CC Outputs/Current setpoint value Ch.18 <-> Data Pointer/CurrentSetpointValues[17]
//     Term 35 (AT2200-0500)/CC Outputs/Current setpoint value Ch.19 <-> Data Pointer/CurrentSetpointValues[18]
//     Term 35 (AT2200-0500)/CC Outputs/Current setpoint value Ch.2 <-> Data Pointer/CurrentSetpointValues[1]
//     Term 35 (AT2200-0500)/CC Outputs/Current setpoint value Ch.20 <-> Data Pointer/CurrentSetpointValues[19]
//     Term 35 (AT2200-0500)/CC Outputs/Current setpoint value Ch.21 <-> Data Pointer/CurrentSetpointValues[20]
//     Term 35 (AT2200-0500)/CC Outputs/Current setpoint value Ch.22 <-> Data Pointer/CurrentSetpointValues[21]
//     Term 35 (AT2200-0500)/CC Outputs/Current setpoint value Ch.23 <-> Data Pointer/CurrentSetpointValues[22]
//     Term 35 (AT2200-0500)/CC Outputs/Current setpoint value Ch.24 <-> Data Pointer/CurrentSetpointValues[23]
//     Term 35 (AT2200-0500)/CC Outputs/Current setpoint value Ch.25 <-> Data Pointer/CurrentSetpointValues[24]
//     Term 35 (AT2200-0500)/CC Outputs/Current setpoint value Ch.26 <-> Data Pointer/CurrentSetpointValues[25]
//     Term 35 (AT2200-0500)/CC Outputs/Current setpoint value Ch.27 <-> Data Pointer/CurrentSetpointValues[26]
//     Term 35 (AT2200-0500)/CC Outputs/Current setpoint value Ch.28 <-> Data Pointer/CurrentSetpointValues[27]
//     Term 35 (AT2200-0500)/CC Outputs/Current setpoint value Ch.29 <-> Data Pointer/CurrentSetpointValues[28]
//     Term 35 (AT2200-0500)/CC Outputs/Current setpoint value Ch.3 <-> Data Pointer/CurrentSetpointValues[2]
//     Term 35 (AT2200-0500)/CC Outputs/Current setpoint value Ch.30 <-> Data Pointer/CurrentSetpointValues[29]
//     Term 35 (AT2200-0500)/CC Outputs/Current setpoint value Ch.4 <-> Data Pointer/CurrentSetpointValues[3]
//     Term 35 (AT2200-0500)/CC Outputs/Current setpoint value Ch.5 <-> Data Pointer/CurrentSetpointValues[4]
//     Term 35 (AT2200-0500)/CC Outputs/Current setpoint value Ch.6 <-> Data Pointer/CurrentSetpointValues[5]
//     Term 35 (AT2200-0500)/CC Outputs/Current setpoint value Ch.7 <-> Data Pointer/CurrentSetpointValues[6]
//     Term 35 (AT2200-0500)/CC Outputs/Current setpoint value Ch.8 <-> Data Pointer/CurrentSetpointValues[7]
//     Term 35 (AT2200-0500)/CC Outputs/Current setpoint value Ch.9 <-> Data Pointer/CurrentSetpointValues[8]
//     Term 35 (AT2200-0500)/LFB Inputs/BinaryData <-> Data Pointer/HallSensorValues
//   Device 24 <-> TcCOM Objects/XTS ProcessingUnit 1/Part 1/Module 28
//     Term 36 (AT2200-0500)/CC Inputs/Current actual value Ch.1 <-> Data Pointer/CurrentActualValues[0]
//     Term 36 (AT2200-0500)/CC Inputs/Current actual value Ch.10 <-> Data Pointer/CurrentActualValues[9]
//     Term 36 (AT2200-0500)/CC Inputs/Current actual value Ch.11 <-> Data Pointer/CurrentActualValues[10]
//     Term 36 (AT2200-0500)/CC Inputs/Current actual value Ch.12 <-> Data Pointer/CurrentActualValues[11]
//     Term 36 (AT2200-0500)/CC Inputs/Current actual value Ch.13 <-> Data Pointer/CurrentActualValues[12]
//     Term 36 (AT2200-0500)/CC Inputs/Current actual value Ch.14 <-> Data Pointer/CurrentActualValues[13]
//     Term 36 (AT2200-0500)/CC Inputs/Current actual value Ch.15 <-> Data Pointer/CurrentActualValues[14]
//     Term 36 (AT2200-0500)/CC Inputs/Current actual value Ch.16 <-> Data Pointer/CurrentActualValues[15]
//     Term 36 (AT2200-0500)/CC Inputs/Current actual value Ch.17 <-> Data Pointer/CurrentActualValues[16]
//     Term 36 (AT2200-0500)/CC Inputs/Current actual value Ch.18 <-> Data Pointer/CurrentActualValues[17]
//     Term 36 (AT2200-0500)/CC Inputs/Current actual value Ch.19 <-> Data Pointer/CurrentActualValues[18]
//     Term 36 (AT2200-0500)/CC Inputs/Current actual value Ch.2 <-> Data Pointer/CurrentActualValues[1]
//     Term 36 (AT2200-0500)/CC Inputs/Current actual value Ch.20 <-> Data Pointer/CurrentActualValues[19]
//     Term 36 (AT2200-0500)/CC Inputs/Current actual value Ch.21 <-> Data Pointer/CurrentActualValues[20]
//     Term 36 (AT2200-0500)/CC Inputs/Current actual value Ch.22 <-> Data Pointer/CurrentActualValues[21]
//     Term 36 (AT2200-0500)/CC Inputs/Current actual value Ch.23 <-> Data Pointer/CurrentActualValues[22]
//     Term 36 (AT2200-0500)/CC Inputs/Current actual value Ch.24 <-> Data Pointer/CurrentActualValues[23]
//     Term 36 (AT2200-0500)/CC Inputs/Current actual value Ch.25 <-> Data Pointer/CurrentActualValues[24]
//     Term 36 (AT2200-0500)/CC Inputs/Current actual value Ch.26 <-> Data Pointer/CurrentActualValues[25]
//     Term 36 (AT2200-0500)/CC Inputs/Current actual value Ch.27 <-> Data Pointer/CurrentActualValues[26]
//     Term 36 (AT2200-0500)/CC Inputs/Current actual value Ch.28 <-> Data Pointer/CurrentActualValues[27]
//     Term 36 (AT2200-0500)/CC Inputs/Current actual value Ch.29 <-> Data Pointer/CurrentActualValues[28]
//     Term 36 (AT2200-0500)/CC Inputs/Current actual value Ch.3 <-> Data Pointer/CurrentActualValues[2]
//     Term 36 (AT2200-0500)/CC Inputs/Current actual value Ch.30 <-> Data Pointer/CurrentActualValues[29]
//     Term 36 (AT2200-0500)/CC Inputs/Current actual value Ch.4 <-> Data Pointer/CurrentActualValues[3]
//     Term 36 (AT2200-0500)/CC Inputs/Current actual value Ch.5 <-> Data Pointer/CurrentActualValues[4]
//     Term 36 (AT2200-0500)/CC Inputs/Current actual value Ch.6 <-> Data Pointer/CurrentActualValues[5]
//     Term 36 (AT2200-0500)/CC Inputs/Current actual value Ch.7 <-> Data Pointer/CurrentActualValues[6]
//     Term 36 (AT2200-0500)/CC Inputs/Current actual value Ch.8 <-> Data Pointer/CurrentActualValues[7]
//     Term 36 (AT2200-0500)/CC Inputs/Current actual value Ch.9 <-> Data Pointer/CurrentActualValues[8]
//     Term 36 (AT2200-0500)/CC Inputs/Status <-> Data Pointer/Status
//     Term 36 (AT2200-0500)/CC Outputs/Control <-> Data Pointer/Control
//     Term 36 (AT2200-0500)/CC Outputs/Current setpoint value Ch.1 <-> Data Pointer/CurrentSetpointValues[0]
//     Term 36 (AT2200-0500)/CC Outputs/Current setpoint value Ch.10 <-> Data Pointer/CurrentSetpointValues[9]
//     Term 36 (AT2200-0500)/CC Outputs/Current setpoint value Ch.11 <-> Data Pointer/CurrentSetpointValues[10]
//     Term 36 (AT2200-0500)/CC Outputs/Current setpoint value Ch.12 <-> Data Pointer/CurrentSetpointValues[11]
//     Term 36 (AT2200-0500)/CC Outputs/Current setpoint value Ch.13 <-> Data Pointer/CurrentSetpointValues[12]
//     Term 36 (AT2200-0500)/CC Outputs/Current setpoint value Ch.14 <-> Data Pointer/CurrentSetpointValues[13]
//     Term 36 (AT2200-0500)/CC Outputs/Current setpoint value Ch.15 <-> Data Pointer/CurrentSetpointValues[14]
//     Term 36 (AT2200-0500)/CC Outputs/Current setpoint value Ch.16 <-> Data Pointer/CurrentSetpointValues[15]
//     Term 36 (AT2200-0500)/CC Outputs/Current setpoint value Ch.17 <-> Data Pointer/CurrentSetpointValues[16]
//     Term 36 (AT2200-0500)/CC Outputs/Current setpoint value Ch.18 <-> Data Pointer/CurrentSetpointValues[17]
//     Term 36 (AT2200-0500)/CC Outputs/Current setpoint value Ch.19 <-> Data Pointer/CurrentSetpointValues[18]
//     Term 36 (AT2200-0500)/CC Outputs/Current setpoint value Ch.2 <-> Data Pointer/CurrentSetpointValues[1]
//     Term 36 (AT2200-0500)/CC Outputs/Current setpoint value Ch.20 <-> Data Pointer/CurrentSetpointValues[19]
//     Term 36 (AT2200-0500)/CC Outputs/Current setpoint value Ch.21 <-> Data Pointer/CurrentSetpointValues[20]
//     Term 36 (AT2200-0500)/CC Outputs/Current setpoint value Ch.22 <-> Data Pointer/CurrentSetpointValues[21]
//     Term 36 (AT2200-0500)/CC Outputs/Current setpoint value Ch.23 <-> Data Pointer/CurrentSetpointValues[22]
//     Term 36 (AT2200-0500)/CC Outputs/Current setpoint value Ch.24 <-> Data Pointer/CurrentSetpointValues[23]
//     Term 36 (AT2200-0500)/CC Outputs/Current setpoint value Ch.25 <-> Data Pointer/CurrentSetpointValues[24]
//     Term 36 (AT2200-0500)/CC Outputs/Current setpoint value Ch.26 <-> Data Pointer/CurrentSetpointValues[25]
//     Term 36 (AT2200-0500)/CC Outputs/Current setpoint value Ch.27 <-> Data Pointer/CurrentSetpointValues[26]
//     Term 36 (AT2200-0500)/CC Outputs/Current setpoint value Ch.28 <-> Data Pointer/CurrentSetpointValues[27]
//     Term 36 (AT2200-0500)/CC Outputs/Current setpoint value Ch.29 <-> Data Pointer/CurrentSetpointValues[28]
//     Term 36 (AT2200-0500)/CC Outputs/Current setpoint value Ch.3 <-> Data Pointer/CurrentSetpointValues[2]
//     Term 36 (AT2200-0500)/CC Outputs/Current setpoint value Ch.30 <-> Data Pointer/CurrentSetpointValues[29]
//     Term 36 (AT2200-0500)/CC Outputs/Current setpoint value Ch.4 <-> Data Pointer/CurrentSetpointValues[3]
//     Term 36 (AT2200-0500)/CC Outputs/Current setpoint value Ch.5 <-> Data Pointer/CurrentSetpointValues[4]
//     Term 36 (AT2200-0500)/CC Outputs/Current setpoint value Ch.6 <-> Data Pointer/CurrentSetpointValues[5]
//     Term 36 (AT2200-0500)/CC Outputs/Current setpoint value Ch.7 <-> Data Pointer/CurrentSetpointValues[6]
//     Term 36 (AT2200-0500)/CC Outputs/Current setpoint value Ch.8 <-> Data Pointer/CurrentSetpointValues[7]
//     Term 36 (AT2200-0500)/CC Outputs/Current setpoint value Ch.9 <-> Data Pointer/CurrentSetpointValues[8]
//     Term 36 (AT2200-0500)/LFB Inputs/BinaryData <-> Data Pointer/HallSensorValues
//   Device 25 <-> TcCOM Objects/XTS ProcessingUnit 1/Part 1/Module 29
//     Term 37 (AT2202-0500)/CC Inputs/Current actual value Ch.1 <-> Data Pointer/CurrentActualValues[0]
//     Term 37 (AT2202-0500)/CC Inputs/Current actual value Ch.10 <-> Data Pointer/CurrentActualValues[9]
//     Term 37 (AT2202-0500)/CC Inputs/Current actual value Ch.11 <-> Data Pointer/CurrentActualValues[10]
//     Term 37 (AT2202-0500)/CC Inputs/Current actual value Ch.12 <-> Data Pointer/CurrentActualValues[11]
//     Term 37 (AT2202-0500)/CC Inputs/Current actual value Ch.13 <-> Data Pointer/CurrentActualValues[12]
//     Term 37 (AT2202-0500)/CC Inputs/Current actual value Ch.14 <-> Data Pointer/CurrentActualValues[13]
//     Term 37 (AT2202-0500)/CC Inputs/Current actual value Ch.15 <-> Data Pointer/CurrentActualValues[14]
//     Term 37 (AT2202-0500)/CC Inputs/Current actual value Ch.16 <-> Data Pointer/CurrentActualValues[15]
//     Term 37 (AT2202-0500)/CC Inputs/Current actual value Ch.17 <-> Data Pointer/CurrentActualValues[16]
//     Term 37 (AT2202-0500)/CC Inputs/Current actual value Ch.18 <-> Data Pointer/CurrentActualValues[17]
//     Term 37 (AT2202-0500)/CC Inputs/Current actual value Ch.19 <-> Data Pointer/CurrentActualValues[18]
//     Term 37 (AT2202-0500)/CC Inputs/Current actual value Ch.2 <-> Data Pointer/CurrentActualValues[1]
//     Term 37 (AT2202-0500)/CC Inputs/Current actual value Ch.20 <-> Data Pointer/CurrentActualValues[19]
//     Term 37 (AT2202-0500)/CC Inputs/Current actual value Ch.21 <-> Data Pointer/CurrentActualValues[20]
//     Term 37 (AT2202-0500)/CC Inputs/Current actual value Ch.22 <-> Data Pointer/CurrentActualValues[21]
//     Term 37 (AT2202-0500)/CC Inputs/Current actual value Ch.23 <-> Data Pointer/CurrentActualValues[22]
//     Term 37 (AT2202-0500)/CC Inputs/Current actual value Ch.24 <-> Data Pointer/CurrentActualValues[23]
//     Term 37 (AT2202-0500)/CC Inputs/Current actual value Ch.25 <-> Data Pointer/CurrentActualValues[24]
//     Term 37 (AT2202-0500)/CC Inputs/Current actual value Ch.26 <-> Data Pointer/CurrentActualValues[25]
//     Term 37 (AT2202-0500)/CC Inputs/Current actual value Ch.27 <-> Data Pointer/CurrentActualValues[26]
//     Term 37 (AT2202-0500)/CC Inputs/Current actual value Ch.28 <-> Data Pointer/CurrentActualValues[27]
//     Term 37 (AT2202-0500)/CC Inputs/Current actual value Ch.29 <-> Data Pointer/CurrentActualValues[28]
//     Term 37 (AT2202-0500)/CC Inputs/Current actual value Ch.3 <-> Data Pointer/CurrentActualValues[2]
//     Term 37 (AT2202-0500)/CC Inputs/Current actual value Ch.30 <-> Data Pointer/CurrentActualValues[29]
//     Term 37 (AT2202-0500)/CC Inputs/Current actual value Ch.4 <-> Data Pointer/CurrentActualValues[3]
//     Term 37 (AT2202-0500)/CC Inputs/Current actual value Ch.5 <-> Data Pointer/CurrentActualValues[4]
//     Term 37 (AT2202-0500)/CC Inputs/Current actual value Ch.6 <-> Data Pointer/CurrentActualValues[5]
//     Term 37 (AT2202-0500)/CC Inputs/Current actual value Ch.7 <-> Data Pointer/CurrentActualValues[6]
//     Term 37 (AT2202-0500)/CC Inputs/Current actual value Ch.8 <-> Data Pointer/CurrentActualValues[7]
//     Term 37 (AT2202-0500)/CC Inputs/Current actual value Ch.9 <-> Data Pointer/CurrentActualValues[8]
//     Term 37 (AT2202-0500)/CC Inputs/Status <-> Data Pointer/Status
//     Term 37 (AT2202-0500)/CC Outputs/Control <-> Data Pointer/Control
//     Term 37 (AT2202-0500)/CC Outputs/Current setpoint value Ch.1 <-> Data Pointer/CurrentSetpointValues[0]
//     Term 37 (AT2202-0500)/CC Outputs/Current setpoint value Ch.10 <-> Data Pointer/CurrentSetpointValues[9]
//     Term 37 (AT2202-0500)/CC Outputs/Current setpoint value Ch.11 <-> Data Pointer/CurrentSetpointValues[10]
//     Term 37 (AT2202-0500)/CC Outputs/Current setpoint value Ch.12 <-> Data Pointer/CurrentSetpointValues[11]
//     Term 37 (AT2202-0500)/CC Outputs/Current setpoint value Ch.13 <-> Data Pointer/CurrentSetpointValues[12]
//     Term 37 (AT2202-0500)/CC Outputs/Current setpoint value Ch.14 <-> Data Pointer/CurrentSetpointValues[13]
//     Term 37 (AT2202-0500)/CC Outputs/Current setpoint value Ch.15 <-> Data Pointer/CurrentSetpointValues[14]
//     Term 37 (AT2202-0500)/CC Outputs/Current setpoint value Ch.16 <-> Data Pointer/CurrentSetpointValues[15]
//     Term 37 (AT2202-0500)/CC Outputs/Current setpoint value Ch.17 <-> Data Pointer/CurrentSetpointValues[16]
//     Term 37 (AT2202-0500)/CC Outputs/Current setpoint value Ch.18 <-> Data Pointer/CurrentSetpointValues[17]
//     Term 37 (AT2202-0500)/CC Outputs/Current setpoint value Ch.19 <-> Data Pointer/CurrentSetpointValues[18]
//     Term 37 (AT2202-0500)/CC Outputs/Current setpoint value Ch.2 <-> Data Pointer/CurrentSetpointValues[1]
//     Term 37 (AT2202-0500)/CC Outputs/Current setpoint value Ch.20 <-> Data Pointer/CurrentSetpointValues[19]
//     Term 37 (AT2202-0500)/CC Outputs/Current setpoint value Ch.21 <-> Data Pointer/CurrentSetpointValues[20]
//     Term 37 (AT2202-0500)/CC Outputs/Current setpoint value Ch.22 <-> Data Pointer/CurrentSetpointValues[21]
//     Term 37 (AT2202-0500)/CC Outputs/Current setpoint value Ch.23 <-> Data Pointer/CurrentSetpointValues[22]
//     Term 37 (AT2202-0500)/CC Outputs/Current setpoint value Ch.24 <-> Data Pointer/CurrentSetpointValues[23]
//     Term 37 (AT2202-0500)/CC Outputs/Current setpoint value Ch.25 <-> Data Pointer/CurrentSetpointValues[24]
//     Term 37 (AT2202-0500)/CC Outputs/Current setpoint value Ch.26 <-> Data Pointer/CurrentSetpointValues[25]
//     Term 37 (AT2202-0500)/CC Outputs/Current setpoint value Ch.27 <-> Data Pointer/CurrentSetpointValues[26]
//     Term 37 (AT2202-0500)/CC Outputs/Current setpoint value Ch.28 <-> Data Pointer/CurrentSetpointValues[27]
//     Term 37 (AT2202-0500)/CC Outputs/Current setpoint value Ch.29 <-> Data Pointer/CurrentSetpointValues[28]
//     Term 37 (AT2202-0500)/CC Outputs/Current setpoint value Ch.3 <-> Data Pointer/CurrentSetpointValues[2]
//     Term 37 (AT2202-0500)/CC Outputs/Current setpoint value Ch.30 <-> Data Pointer/CurrentSetpointValues[29]
//     Term 37 (AT2202-0500)/CC Outputs/Current setpoint value Ch.4 <-> Data Pointer/CurrentSetpointValues[3]
//     Term 37 (AT2202-0500)/CC Outputs/Current setpoint value Ch.5 <-> Data Pointer/CurrentSetpointValues[4]
//     Term 37 (AT2202-0500)/CC Outputs/Current setpoint value Ch.6 <-> Data Pointer/CurrentSetpointValues[5]
//     Term 37 (AT2202-0500)/CC Outputs/Current setpoint value Ch.7 <-> Data Pointer/CurrentSetpointValues[6]
//     Term 37 (AT2202-0500)/CC Outputs/Current setpoint value Ch.8 <-> Data Pointer/CurrentSetpointValues[7]
//     Term 37 (AT2202-0500)/CC Outputs/Current setpoint value Ch.9 <-> Data Pointer/CurrentSetpointValues[8]
//     Term 37 (AT2202-0500)/LFB Inputs/BinaryData <-> Data Pointer/HallSensorValues
//   Device 25 <-> TcCOM Objects/XTS ProcessingUnit 1/Part 1/Module 30
//     Term 38 (AT2200-0500)/CC Inputs/Current actual value Ch.1 <-> Data Pointer/CurrentActualValues[0]
//     Term 38 (AT2200-0500)/CC Inputs/Current actual value Ch.10 <-> Data Pointer/CurrentActualValues[9]
//     Term 38 (AT2200-0500)/CC Inputs/Current actual value Ch.11 <-> Data Pointer/CurrentActualValues[10]
//     Term 38 (AT2200-0500)/CC Inputs/Current actual value Ch.12 <-> Data Pointer/CurrentActualValues[11]
//     Term 38 (AT2200-0500)/CC Inputs/Current actual value Ch.13 <-> Data Pointer/CurrentActualValues[12]
//     Term 38 (AT2200-0500)/CC Inputs/Current actual value Ch.14 <-> Data Pointer/CurrentActualValues[13]
//     Term 38 (AT2200-0500)/CC Inputs/Current actual value Ch.15 <-> Data Pointer/CurrentActualValues[14]
//     Term 38 (AT2200-0500)/CC Inputs/Current actual value Ch.16 <-> Data Pointer/CurrentActualValues[15]
//     Term 38 (AT2200-0500)/CC Inputs/Current actual value Ch.17 <-> Data Pointer/CurrentActualValues[16]
//     Term 38 (AT2200-0500)/CC Inputs/Current actual value Ch.18 <-> Data Pointer/CurrentActualValues[17]
//     Term 38 (AT2200-0500)/CC Inputs/Current actual value Ch.19 <-> Data Pointer/CurrentActualValues[18]
//     Term 38 (AT2200-0500)/CC Inputs/Current actual value Ch.2 <-> Data Pointer/CurrentActualValues[1]
//     Term 38 (AT2200-0500)/CC Inputs/Current actual value Ch.20 <-> Data Pointer/CurrentActualValues[19]
//     Term 38 (AT2200-0500)/CC Inputs/Current actual value Ch.21 <-> Data Pointer/CurrentActualValues[20]
//     Term 38 (AT2200-0500)/CC Inputs/Current actual value Ch.22 <-> Data Pointer/CurrentActualValues[21]
//     Term 38 (AT2200-0500)/CC Inputs/Current actual value Ch.23 <-> Data Pointer/CurrentActualValues[22]
//     Term 38 (AT2200-0500)/CC Inputs/Current actual value Ch.24 <-> Data Pointer/CurrentActualValues[23]
//     Term 38 (AT2200-0500)/CC Inputs/Current actual value Ch.25 <-> Data Pointer/CurrentActualValues[24]
//     Term 38 (AT2200-0500)/CC Inputs/Current actual value Ch.26 <-> Data Pointer/CurrentActualValues[25]
//     Term 38 (AT2200-0500)/CC Inputs/Current actual value Ch.27 <-> Data Pointer/CurrentActualValues[26]
//     Term 38 (AT2200-0500)/CC Inputs/Current actual value Ch.28 <-> Data Pointer/CurrentActualValues[27]
//     Term 38 (AT2200-0500)/CC Inputs/Current actual value Ch.29 <-> Data Pointer/CurrentActualValues[28]
//     Term 38 (AT2200-0500)/CC Inputs/Current actual value Ch.3 <-> Data Pointer/CurrentActualValues[2]
